LIN {X 0,Y 418.284,Z 298.384,A -85,B 0,C 180,E1 -10098.617,E2 -10098.617} C_VEL
LIN {X 0,Y 418.234,Z 298.38,A -85,B 0,C 180,E1 -10101.696,E2 -10101.696} C_VEL
LIN {X 0,Y 418.285,Z 298.377,A -85,B 0,C 180,E1 -10104.864,E2 -10104.864} C_VEL
LIN {X 0,Y 418.292,Z 298.377,A -85,B 0,C 180,E1 -10108.063,E2 -10108.063} C_VEL
LIN {X 0,Y 418.212,Z 298.39,A -85,B 0,C 180,E1 -10111.396,E2 -10111.396} C_VEL
LIN {X 0,Y 418.265,Z 298.378,A -85,B 0,C 180,E1 -10114.58,E2 -10114.58} C_VEL
LIN {X 0,Y 418.228,Z 298.385,A -85,B 0,C 180,E1 -10117.833,E2 -10117.833} C_VEL
LIN {X 0,Y 418.223,Z 298.387,A -85,B 0,C 180,E1 -10120.948,E2 -10120.948} C_VEL
LIN {X 0,Y 418.211,Z 298.392,A -85,B 0,C 180,E1 -10123.729,E2 -10123.729} C_VEL
LIN {X 0,Y 418.21,Z 298.388,A -85,B 0,C 180,E1 -10126.449,E2 -10126.449} C_VEL
LIN {X 0,Y 418.225,Z 298.389,A -85,B 0,C 180,E1 -10129.13,E2 -10129.13} C_VEL
LIN {X 0,Y 418.228,Z 298.39,A -85,B 0,C 180,E1 -10132.167,E2 -10132.167} C_VEL
LIN {X 0,Y 418.268,Z 298.385,A -85,B 0,C 180,E1 -10135.42,E2 -10135.42} C_VEL
LIN {X 0,Y 418.214,Z 298.387,A -85,B 0,C 180,E1 -10138.604,E2 -10138.604} C_VEL
LIN {X 0,Y 418.318,Z 298.464,A -85,B 0,C 180,E1 -10141.802,E2 -10141.802} C_VEL
LIN {X 0,Y 420.837,Z 310.121,A -85,B 0,C 180,E1 -10144.397,E2 -10144.397} C_VEL
LIN {X 0,Y 421.67,Z 315.968,A -85,B 0,C 180,E1 -10145.637,E2 -10145.637} C_VEL
LIN {X 0,Y 420.417,Z 334.149,A -85,B 0,C 180,E1 -10149.192,E2 -10149.192} C_VEL
LIN {X 0,Y 419.964,Z 341.407,A -85,B 0,C 180,E1 -10150.586,E2 -10150.586} C_VEL
LIN {X 0,Y 423.935,Z 364.685,A -85,B 0,C 180,E1 -10151.22,E2 -10151.22} C_VEL
LIN {X 0,Y 424.4,Z 369.391,A -85,B 0,C 180,E1 -10151.329,E2 -10151.329} C_VEL
LIN {X 0,Y 423.4,Z 449.942,A -85,B 0,C 180,E1 -10152.74,E2 -10152.74} C_VEL
LIN {X 0,Y 422.877,Z 463.116,A -85,B 0,C 180,E1 -10153.153,E2 -10153.153} C_VEL
LIN {X 0,Y 422.172,Z 475.789,A -85,B 0,C 180,E1 -10153.746,E2 -10153.746} C_VEL
LIN {X 0,Y 421.379,Z 487.877,A -85,B 0,C 180,E1 -10154.522,E2 -10154.522} C_VEL
LIN {X 0,Y 420.519,Z 499.381,A -85,B 0,C 180,E1 -10155.481,E2 -10155.481} C_VEL
LIN {X 0,Y 419.752,Z 509.766,A -85,B 0,C 180,E1 -10156.566,E2 -10156.566} C_VEL
LIN {X 0,Y 419.108,Z 518.281,A -85,B 0,C 180,E1 -10157.654,E2 -10157.654} C_VEL
LIN {X 0,Y 418.408,Z 526.153,A -85,B 0,C 180,E1 -10158.862,E2 -10158.862} C_VEL
LIN {X 0,Y 417.839,Z 533.861,A -85,B 0,C 180,E1 -10160.316,E2 -10160.316} C_VEL
LIN {X 0,Y 417.462,Z 540.067,A -85,B 0,C 180,E1 -10161.772,E2 -10161.772} C_VEL
LIN {X 0,Y 417.234,Z 545.013,A -85,B 0,C 180,E1 -10163.228,E2 -10163.228} C_VEL
LIN {X 0,Y 417.121,Z 548.84,A -85,B 0,C 180,E1 -10164.682,E2 -10164.682} C_VEL
LIN {X 0,Y 417.015,Z 551.649,A -85,B 0,C 180,E1 -10166.134,E2 -10166.134} C_VEL
LIN {X 0,Y 417.069,Z 553.924,A -85,B 0,C 180,E1 -10168.068,E2 -10168.068} C_VEL
LIN {X 0,Y 417.013,Z 554.464,A -85,B 0,C 180,E1 -10169.034,E2 -10169.034} C_VEL
LIN {X 0,Y 417.027,Z 554.573,A -85,B 0,C 180,E1 -10169.999,E2 -10169.999} C_VEL
LIN {X 0,Y 417.072,Z 553.622,A -85,B 0,C 180,E1 -10171.931,E2 -10171.931} C_VEL
LIN {X 0,Y 417.06,Z 552.553,A -85,B 0,C 180,E1 -10172.897,E2 -10172.897} C_VEL
LIN {X 0,Y 417.017,Z 551.024,A -85,B 0,C 180,E1 -10173.865,E2 -10173.865} C_VEL
LIN {X 0,Y 417.12,Z 547.943,A -85,B 0,C 180,E1 -10175.316,E2 -10175.316} C_VEL
LIN {X 0,Y 417.23,Z 543.788,A -85,B 0,C 180,E1 -10176.771,E2 -10176.771} C_VEL
LIN {X 0,Y 417.492,Z 537.427,A -85,B 0,C 180,E1 -10178.469,E2 -10178.469} C_VEL
LIN {X 0,Y 417.857,Z 530.492,A -85,B 0,C 180,E1 -10179.926,E2 -10179.926} C_VEL
LIN {X 0,Y 418.284,Z 523.404,A -85,B 0,C 180,E1 -10181.14,E2 -10181.14} C_VEL
LIN {X 0,Y 418.883,Z 514.854,A -85,B 0,C 180,E1 -10182.351,E2 -10182.351} C_VEL
LIN {X 0,Y 419.561,Z 504.271,A -85,B 0,C 180,E1 -10183.562,E2 -10183.562} C_VEL
LIN {X 0,Y 420.202,Z 493.786,A -85,B 0,C 180,E1 -10184.529,E2 -10184.529} C_VEL
LIN {X 0,Y 420.853,Z 482.263,A -85,B 0,C 180,E1 -10185.372,E2 -10185.372} C_VEL
LIN {X 0,Y 421.525,Z 470.346,A -85,B 0,C 180,E1 -10186.029,E2 -10186.029} C_VEL
LIN {X 0,Y 421.993,Z 458.396,A -85,B 0,C 180,E1 -10186.508,E2 -10186.508} C_VEL
LIN {X 0,Y 422.351,Z 445.617,A -85,B 0,C 180,E1 -10186.836,E2 -10186.836} C_VEL
LIN {X 0,Y 423.12,Z 367.397,A -85,B 0,C 180,E1 -10188.171,E2 -10188.171} C_VEL
LIN {X 0,Y 419.362,Z 341.793,A -85,B 0,C 180,E1 -10188.764,E2 -10188.764} C_VEL
LIN {X 0,Y 420.312,Z 325.648,A -85,B 0,C 180,E1 -10191.84,E2 -10191.84} C_VEL
LIN {X 0,Y 421.019,Z 313.701,A -85,B 0,C 180,E1 -10194.139,E2 -10194.139} C_VEL
LIN {X 0,Y 419.772,Z 305.575,A -85,B 0,C 180,E1 -10195.803,E2 -10195.803} C_VEL
LIN {X 0,Y 418.343,Z 298.377,A -85,B 0,C 180,E1 -10197.328,E2 -10197.328} C_VEL
LIN {X 0,Y 418.236,Z 298.384,A -85,B 0,C 180,E1 -10201.019,E2 -10201.019} C_VEL
LIN {X 0,Y 418.246,Z 298.384,A -85,B 0,C 180,E1 -10203.676,E2 -10203.676} C_VEL
LIN {X 0,Y 418.236,Z 298.383,A -85,B 0,C 180,E1 -10207.223,E2 -10207.223} C_VEL
LIN {X 0,Y 418.24,Z 298.383,A -85,B 0,C 180,E1 -10209.682,E2 -10209.682} C_VEL
LIN {X 0,Y 418.225,Z 298.391,A -85,B 0,C 180,E1 -10212.32,E2 -10212.32} C_VEL
LIN {X 0,Y 418.234,Z 298.384,A -85,B 0,C 180,E1 -10215.108,E2 -10215.108} C_VEL
LIN {X 0,Y 418.237,Z 298.383,A -85,B 0,C 180,E1 -10217.766,E2 -10217.766} C_VEL
LIN {X 0,Y 418.254,Z 298.389,A -85,B 0,C 180,E1 -10220.617,E2 -10220.617} C_VEL
LIN {X 0,Y 418.239,Z 298.383,A -85,B 0,C 180,E1 -10223.975,E2 -10223.975} C_VEL
LIN {X 0,Y 418.254,Z 298.384,A -85,B 0,C 180,E1 -10227.155,E2 -10227.155} C_VEL
LIN {X 0,Y 418.268,Z 298.386,A -85,B 0,C 180,E1 -10230.838,E2 -10230.838} C_VEL
LIN {X 0,Y 418.263,Z 298.38,A -85,B 0,C 180,E1 -10234.095,E2 -10234.095} C_VEL
LIN {X 0,Y 418.229,Z 298.389,A -85,B 0,C 180,E1 -10237.263,E2 -10237.263} C_VEL
LIN {X 0,Y 418.274,Z 298.378,A -85,B 0,C 180,E1 -10240.364,E2 -10240.364} C_VEL
LIN {X 0,Y 418.308,Z 298.38,A -85,B 0,C 180,E1 -10243.404,E2 -10243.404} C_VEL
LIN {X 0,Y 418.337,Z 298.374,A -85,B 0,C 180,E1 -10246.999,E2 -10246.999} C_VEL
LIN {X 0,Y 418.333,Z 298.371,A -85,B 0,C 180,E1 -10250.328,E2 -10250.328} C_VEL
LIN {X 0,Y 418.504,Z 298.35,A -85,B 0,C 180,E1 -10252.279,E2 -10252.279} C_VEL
LIN {X 0,Y 418.503,Z 298.35,A -85,B 0,C 180,E1 -10254.217,E2 -10254.217} C_VEL
LIN {X 0,Y 418.534,Z 298.348,A -85,B 0,C 180,E1 -10258.075,E2 -10258.075} C_VEL
LIN {X 0,Y 418.662,Z 298.334,A -85,B 0,C 180,E1 -10260,E2 -10260} C_VEL
LIN {X 0,Y 418.501,Z 298.35,A -85,B 0,C 180,E1 -10262.888,E2 -10262.888} C_VEL
LIN {X 0,Y 418.448,Z 298.357,A -85,B 0,C 180,E1 -10266.523,E2 -10266.523} C_VEL
LIN {X 0,Y 418.331,Z 298.376,A -85,B 0,C 180,E1 -10269.672,E2 -10269.672} C_VEL
LIN {X 0,Y 418.337,Z 298.37,A -85,B 0,C 180,E1 -10273.001,E2 -10273.001} C_VEL
LIN {X 0,Y 418.311,Z 298.375,A -85,B 0,C 180,E1 -10276.739,E2 -10276.739} C_VEL
LIN {X 0,Y 418.262,Z 298.383,A -85,B 0,C 180,E1 -10279.791,E2 -10279.791} C_VEL
LIN {X 0,Y 418.223,Z 298.387,A -85,B 0,C 180,E1 -10282.737,E2 -10282.737} C_VEL
LIN {X 0,Y 418.253,Z 298.383,A -85,B 0,C 180,E1 -10285.905,E2 -10285.905} C_VEL
LIN {X 0,Y 418.261,Z 298.381,A -85,B 0,C 180,E1 -10289.105,E2 -10289.105} C_VEL
LIN {X 0,Y 418.25,Z 298.385,A -85,B 0,C 180,E1 -10292.845,E2 -10292.845} C_VEL
LIN {X 0,Y 418.238,Z 298.386,A -85,B 0,C 180,E1 -10296.239,E2 -10296.239} C_VEL
LIN {X 0,Y 418.194,Z 298.388,A -85,B 0,C 180,E1 -10299.689,E2 -10299.689} C_VEL
LIN {X 0,Y 418.215,Z 298.388,A -85,B 0,C 180,E1 -10302.321,E2 -10302.321} C_VEL
LIN {X 0,Y 418.23,Z 298.388,A -85,B 0,C 180,E1 -10305.11,E2 -10305.11} C_VEL
LIN {X 0,Y 418.218,Z 298.385,A -85,B 0,C 180,E1 -10307.766,E2 -10307.766} C_VEL
LIN {X 0,Y 418.236,Z 298.385,A -85,B 0,C 180,E1 -10311.558,E2 -10311.558} C_VEL
LIN {X 0,Y 418.254,Z 298.389,A -85,B 0,C 180,E1 -10315.16,E2 -10315.16} C_VEL
LIN {X 0,Y 418.242,Z 298.387,A -85,B 0,C 180,E1 -10317.473,E2 -10317.473} C_VEL
LIN {X 0,Y 418.257,Z 298.383,A -85,B 0,C 180,E1 -10320.899,E2 -10320.899} C_VEL
LIN {X 0,Y 418.216,Z 298.386,A -85,B 0,C 180,E1 -10324.093,E2 -10324.093} C_VEL
LIN {X 0,Y 418.226,Z 298.389,A -85,B 0,C 180,E1 -10327.264,E2 -10327.264} C_VEL
LIN {X 0,Y 418.283,Z 298.377,A -85,B 0,C 180,E1 -10330.365,E2 -10330.365} C_VEL
LIN {X 0,Y 418.316,Z 298.378,A -85,B 0,C 180,E1 -10333.406,E2 -10333.406} C_VEL
LIN {X 0,Y 418.346,Z 298.37,A -85,B 0,C 180,E1 -10337.001,E2 -10337.001} C_VEL
LIN {X 0,Y 418.318,Z 298.378,A -85,B 0,C 180,E1 -10340.329,E2 -10340.329} C_VEL
LIN {X 0,Y 418.433,Z 298.431,A -85,B 0,C 180,E1 -10342.15,E2 -10342.15} C_VEL
LIN {X 0,Y 419.779,Z 306.465,A -85,B 0,C 180,E1 -10343.994,E2 -10343.994} C_VEL
LIN {X 0,Y 419.625,Z 312.565,A -85,B 0,C 180,E1 -10345.319,E2 -10345.319} C_VEL
LIN {X 0,Y 423.458,Z 333.219,A -85,B 0,C 180,E1 -10345.834,E2 -10345.834} C_VEL
LIN {X 0,Y 422.406,Z 420.671,A -85,B 0,C 180,E1 -10347.346,E2 -10347.346} C_VEL
LIN {X 0,Y 422.186,Z 427.807,A -85,B 0,C 180,E1 -10347.552,E2 -10347.552} C_VEL
LIN {X 0,Y 421.371,Z 433.517,A -85,B 0,C 180,E1 -10347.735,E2 -10347.735} C_VEL
LIN {X 0,Y 418.244,Z 442.663,A -85,B 0,C 180,E1 -10348.05,E2 -10348.05} C_VEL
LIN {X 0,Y 415.058,Z 451.531,A -85,B 0,C 180,E1 -10348.471,E2 -10348.471} C_VEL
LIN {X 0,Y 414.153,Z 456.798,A -85,B 0,C 180,E1 -10348.816,E2 -10348.816} C_VEL
LIN {X 0,Y 413.498,Z 468.178,A -85,B 0,C 180,E1 -10349.757,E2 -10349.757} C_VEL
LIN {X 0,Y 412.779,Z 478.733,A -85,B 0,C 180,E1 -10350.854,E2 -10350.854} C_VEL
LIN {X 0,Y 412.151,Z 487.368,A -85,B 0,C 180,E1 -10351.955,E2 -10351.955} C_VEL
LIN {X 0,Y 411.564,Z 495.326,A -85,B 0,C 180,E1 -10353.182,E2 -10353.182} C_VEL
LIN {X 0,Y 411.026,Z 503.123,A -85,B 0,C 180,E1 -10354.659,E2 -10354.659} C_VEL
LIN {X 0,Y 410.673,Z 509.679,A -85,B 0,C 180,E1 -10356.23,E2 -10356.23} C_VEL
LIN {X 0,Y 410.333,Z 515.036,A -85,B 0,C 180,E1 -10357.876,E2 -10357.876} C_VEL
LIN {X 0,Y 410.103,Z 518.7,A -85,B 0,C 180,E1 -10359.37,E2 -10359.37} C_VEL
LIN {X 0,Y 409.992,Z 521.335,A -85,B 0,C 180,E1 -10360.869,E2 -10360.869} C_VEL
LIN {X 0,Y 409.922,Z 522.9,A -85,B 0,C 180,E1 -10362.244,E2 -10362.244} C_VEL
LIN {X 0,Y 409.815,Z 523.749,A -85,B 0,C 180,E1 -10363.892,E2 -10363.892} C_VEL
LIN {X 0,Y 409.852,Z 523.728,A -85,B 0,C 180,E1 -10364.905,E2 -10364.905} C_VEL
LIN {X 0,Y 409.924,Z 523.045,A -85,B 0,C 180,E1 -10366.239,E2 -10366.239} C_VEL
LIN {X 0,Y 410.002,Z 521.082,A -85,B 0,C 180,E1 -10367.972,E2 -10367.972} C_VEL
LIN {X 0,Y 410.314,Z 518.063,A -85,B 0,C 180,E1 -10369.599,E2 -10369.599} C_VEL
LIN {X 0,Y 410.584,Z 514.287,A -85,B 0,C 180,E1 -10371.067,E2 -10371.067} C_VEL
LIN {X 0,Y 411.065,Z 508.427,A -85,B 0,C 180,E1 -10372.798,E2 -10372.798} C_VEL
LIN {X 0,Y 411.725,Z 501.106,A -85,B 0,C 180,E1 -10374.453,E2 -10374.453} C_VEL
LIN {X 0,Y 412.316,Z 494.236,A -85,B 0,C 180,E1 -10375.709,E2 -10375.709} C_VEL
LIN {X 0,Y 413.089,Z 485.156,A -85,B 0,C 180,E1 -10377.072,E2 -10377.072} C_VEL
LIN {X 0,Y 413.946,Z 475.508,A -85,B 0,C 180,E1 -10378.236,E2 -10378.236} C_VEL
LIN {X 0,Y 414.832,Z 464.643,A -85,B 0,C 180,E1 -10379.288,E2 -10379.288} C_VEL
LIN {X 0,Y 415.607,Z 452.692,A -85,B 0,C 180,E1 -10380.204,E2 -10380.204} C_VEL
LIN {X 0,Y 416.266,Z 440.132,A -85,B 0,C 180,E1 -10380.924,E2 -10380.924} C_VEL
LIN {X 0,Y 416.758,Z 427.18,A -85,B 0,C 180,E1 -10381.448,E2 -10381.448} C_VEL
LIN {X 0,Y 417.031,Z 413.94,A -85,B 0,C 180,E1 -10381.779,E2 -10381.779} C_VEL
LIN {X 0,Y 418.276,Z 334.084,A -85,B 0,C 180,E1 -10383.17,E2 -10383.17} C_VEL
LIN {X 0,Y 414.67,Z 317.421,A -85,B 0,C 180,E1 -10383.684,E2 -10383.684} C_VEL
LIN {X 0,Y 413.565,Z 312.818,A -85,B 0,C 180,E1 -10383.857,E2 -10383.857} C_VEL
LIN {X 0,Y 413.337,Z 308.963,A -85,B 0,C 180,E1 -10384.723,E2 -10384.723} C_VEL
LIN {X 0,Y 411.204,Z 299.261,A -85,B 0,C 180,E1 -10387.085,E2 -10387.085} C_VEL
LIN {X 0,Y 411.182,Z 299.268,A -85,B 0,C 180,E1 -10390.504,E2 -10390.504} C_VEL
LIN {X 0,Y 411.175,Z 299.269,A -85,B 0,C 180,E1 -10393.134,E2 -10393.134} C_VEL
LIN {X 0,Y 411.17,Z 299.269,A -85,B 0,C 180,E1 -10395.881,E2 -10395.881} C_VEL
LIN {X 0,Y 411.167,Z 299.273,A -85,B 0,C 180,E1 -10398.771,E2 -10398.771} C_VEL
LIN {X 0,Y 411.208,Z 299.259,A -85,B 0,C 180,E1 -10401.831,E2 -10401.831} C_VEL
LIN {X 0,Y 411.212,Z 299.265,A -85,B 0,C 180,E1 -10405.121,E2 -10405.121} C_VEL
LIN {X 0,Y 411.167,Z 299.265,A -85,B 0,C 180,E1 -10408.003,E2 -10408.003} C_VEL
LIN {X 0,Y 411.219,Z 299.262,A -85,B 0,C 180,E1 -10411.41,E2 -10411.41} C_VEL
LIN {X 0,Y 411.239,Z 299.257,A -85,B 0,C 180,E1 -10413.619,E2 -10413.619} C_VEL
LIN {X 0,Y 411.204,Z 299.26,A -85,B 0,C 180,E1 -10416.852,E2 -10416.852} C_VEL
LIN {X 0,Y 411.215,Z 299.256,A -85,B 0,C 180,E1 -10420.05,E2 -10420.05} C_VEL
LIN {X 0,Y 411.264,Z 299.255,A -85,B 0,C 180,E1 -10423.131,E2 -10423.131} C_VEL
LIN {X 0,Y 411.306,Z 299.245,A -85,B 0,C 180,E1 -10426.896,E2 -10426.896} C_VEL
LIN {X 0,Y 411.293,Z 299.242,A -85,B 0,C 180,E1 -10430.161,E2 -10430.161} C_VEL
LIN {X 0,Y 411.483,Z 299.228,A -85,B 0,C 180,E1 -10432.147,E2 -10432.147} C_VEL
LIN {X 0,Y 411.472,Z 299.226,A -85,B 0,C 180,E1 -10434.118,E2 -10434.118} C_VEL
LIN {X 0,Y 411.511,Z 299.227,A -85,B 0,C 180,E1 -10438.043,E2 -10438.043} C_VEL
LIN {X 0,Y 411.64,Z 299.203,A -85,B 0,C 180,E1 -10440,E2 -10440} C_VEL
LIN {X 0,Y 411.458,Z 299.227,A -85,B 0,C 180,E1 -10442.937,E2 -10442.937} C_VEL
LIN {X 0,Y 411.458,Z 299.224,A -85,B 0,C 180,E1 -10446.867,E2 -10446.867} C_VEL
LIN {X 0,Y 411.354,Z 299.241,A -85,B 0,C 180,E1 -10448.845,E2 -10448.845} C_VEL
LIN {X 0,Y 411.283,Z 299.242,A -85,B 0,C 180,E1 -10451.833,E2 -10451.833} C_VEL
LIN {X 0,Y 411.26,Z 299.251,A -85,B 0,C 180,E1 -10454.853,E2 -10454.853} C_VEL
LIN {X 0,Y 411.253,Z 299.253,A -85,B 0,C 180,E1 -10457.915,E2 -10457.915} C_VEL
LIN {X 0,Y 411.197,Z 299.258,A -85,B 0,C 180,E1 -10461.034,E2 -10461.034} C_VEL
LIN {X 0,Y 411.221,Z 299.26,A -85,B 0,C 180,E1 -10464.216,E2 -10464.216} C_VEL
LIN {X 0,Y 411.26,Z 299.254,A -85,B 0,C 180,E1 -10467.478,E2 -10467.478} C_VEL
LIN {X 0,Y 411.19,Z 299.261,A -85,B 0,C 180,E1 -10470.848,E2 -10470.848} C_VEL
LIN {X 0,Y 411.205,Z 299.255,A -85,B 0,C 180,E1 -10474.334,E2 -10474.334} C_VEL
LIN {X 0,Y 411.194,Z 299.261,A -85,B 0,C 180,E1 -10477.974,E2 -10477.974} C_VEL
LIN {X 0,Y 411.165,Z 299.268,A -85,B 0,C 180,E1 -10481.228,E2 -10481.228} C_VEL
LIN {X 0,Y 411.177,Z 299.265,A -85,B 0,C 180,E1 -10484.49,E2 -10484.49} C_VEL
LIN {X 0,Y 411.179,Z 299.265,A -85,B 0,C 180,E1 -10488.195,E2 -10488.195} C_VEL
LIN {X 0,Y 411.213,Z 299.255,A -85,B 0,C 180,E1 -10490.775,E2 -10490.775} C_VEL
LIN {X 0,Y 411.2,Z 299.261,A -85,B 0,C 180,E1 -10494.471,E2 -10494.471} C_VEL
LIN {X 0,Y 411.21,Z 299.258,A -85,B 0,C 180,E1 -10496.873,E2 -10496.873} C_VEL
LIN {X 0,Y 411.236,Z 299.258,A -85,B 0,C 180,E1 -10500.644,E2 -10500.644} C_VEL
LIN {X 0,Y 411.283,Z 299.335,A -85,B 0,C 180,E1 -10501.453,E2 -10501.453} C_VEL
LIN {X 0,Y 413.867,Z 311.218,A -85,B 0,C 180,E1 -10504.16,E2 -10504.16} C_VEL
LIN {X 0,Y 414.798,Z 317.271,A -85,B 0,C 180,E1 -10505.473,E2 -10505.473} C_VEL
LIN {X 0,Y 413.555,Z 334.145,A -85,B 0,C 180,E1 -10508.83,E2 -10508.83} C_VEL
LIN {X 0,Y 413.096,Z 341.021,A -85,B 0,C 180,E1 -10510.184,E2 -10510.184} C_VEL
LIN {X 0,Y 417.111,Z 363.869,A -85,B 0,C 180,E1 -10510.841,E2 -10510.841} C_VEL
LIN {X 0,Y 417.802,Z 369.66,A -85,B 0,C 180,E1 -10510.984,E2 -10510.984} C_VEL
LIN {X 0,Y 416.721,Z 450.224,A -85,B 0,C 180,E1 -10512.422,E2 -10512.422} C_VEL
LIN {X 0,Y 416.167,Z 463.217,A -85,B 0,C 180,E1 -10512.842,E2 -10512.842} C_VEL
LIN {X 0,Y 415.405,Z 476.34,A -85,B 0,C 180,E1 -10513.474,E2 -10513.474} C_VEL
LIN {X 0,Y 414.562,Z 488.193,A -85,B 0,C 180,E1 -10514.261,E2 -10514.261} C_VEL
LIN {X 0,Y 413.652,Z 499.591,A -85,B 0,C 180,E1 -10515.235,E2 -10515.235} C_VEL
LIN {X 0,Y 412.832,Z 509.89,A -85,B 0,C 180,E1 -10516.337,E2 -10516.337} C_VEL
LIN {X 0,Y 412.152,Z 518.328,A -85,B 0,C 180,E1 -10517.442,E2 -10517.442} C_VEL
LIN {X 0,Y 411.301,Z 527.498,A -85,B 0,C 180,E1 -10518.916,E2 -10518.916} C_VEL
LIN {X 0,Y 410.744,Z 534.898,A -85,B 0,C 180,E1 -10520.396,E2 -10520.396} C_VEL
LIN {X 0,Y 410.322,Z 541.736,A -85,B 0,C 180,E1 -10522.124,E2 -10522.124} C_VEL
LIN {X 0,Y 410.043,Z 546.698,A -85,B 0,C 180,E1 -10523.774,E2 -10523.774} C_VEL
LIN {X 0,Y 410.018,Z 549.718,A -85,B 0,C 180,E1 -10525.083,E2 -10525.083} C_VEL
LIN {X 0,Y 409.928,Z 552.761,A -85,B 0,C 180,E1 -10527.051,E2 -10527.051} C_VEL
LIN {X 0,Y 409.996,Z 553.691,A -85,B 0,C 180,E1 -10528.035,E2 -10528.035} C_VEL
LIN {X 0,Y 409.938,Z 554.209,A -85,B 0,C 180,E1 -10529.017,E2 -10529.017} C_VEL
LIN {X 0,Y 409.948,Z 554.302,A -85,B 0,C 180,E1 -10529.999,E2 -10529.999} C_VEL
LIN {X 0,Y 410,Z 553.326,A -85,B 0,C 180,E1 -10531.964,E2 -10531.964} C_VEL
LIN {X 0,Y 409.959,Z 552.234,A -85,B 0,C 180,E1 -10532.947,E2 -10532.947} C_VEL
LIN {X 0,Y 409.936,Z 550.687,A -85,B 0,C 180,E1 -10533.931,E2 -10533.931} C_VEL
LIN {X 0,Y 410.017,Z 547.576,A -85,B 0,C 180,E1 -10535.409,E2 -10535.409} C_VEL
LIN {X 0,Y 410.162,Z 543.392,A -85,B 0,C 180,E1 -10536.888,E2 -10536.888} C_VEL
LIN {X 0,Y 410.423,Z 536.996,A -85,B 0,C 180,E1 -10538.616,E2 -10538.616} C_VEL
LIN {X 0,Y 410.799,Z 530.022,A -85,B 0,C 180,E1 -10540.099,E2 -10540.099} C_VEL
LIN {X 0,Y 411.414,Z 521.274,A -85,B 0,C 180,E1 -10541.578,E2 -10541.578} C_VEL
LIN {X 0,Y 412.001,Z 512.298,A -85,B 0,C 180,E1 -10542.811,E2 -10542.811} C_VEL
LIN {X 0,Y 412.648,Z 502.786,A -85,B 0,C 180,E1 -10543.881,E2 -10543.881} C_VEL
LIN {X 0,Y 413.361,Z 491.551,A -85,B 0,C 180,E1 -10544.9,E2 -10544.9} C_VEL
LIN {X 0,Y 414.111,Z 479.331,A -85,B 0,C 180,E1 -10545.755,E2 -10545.755} C_VEL
LIN {X 0,Y 414.783,Z 466.548,A -85,B 0,C 180,E1 -10546.423,E2 -10546.423} C_VEL
LIN {X 0,Y 415.318,Z 453.863,A -85,B 0,C 180,E1 -10546.876,E2 -10546.876} C_VEL
LIN {X 0,Y 415.597,Z 435.872,A -85,B 0,C 180,E1 -10547.244,E2 -10547.244} C_VEL
LIN {X 0,Y 416.181,Z 367.386,A -85,B 0,C 180,E1 -10548.432,E2 -10548.432} C_VEL
LIN {X 0,Y 412.412,Z 341.451,A -85,B 0,C 180,E1 -10549.06,E2 -10549.06} C_VEL
LIN {X 0,Y 413.329,Z 326.457,A -85,B 0,C 180,E1 -10551.966,E2 -10551.966} C_VEL
LIN {X 0,Y 414.035,Z 314.493,A -85,B 0,C 180,E1 -10554.306,E2 -10554.306} C_VEL
LIN {X 0,Y 412.412,Z 304.976,A -85,B 0,C 180,E1 -10556.299,E2 -10556.299} C_VEL
LIN {X 0,Y 411.319,Z 299.251,A -85,B 0,C 180,E1 -10557.541,E2 -10557.541} C_VEL
LIN {X 0,Y 411.18,Z 299.263,A -85,B 0,C 180,E1 -10561.283,E2 -10561.283} C_VEL
LIN {X 0,Y 411.203,Z 299.265,A -85,B 0,C 180,E1 -10564.332,E2 -10564.332} C_VEL
LIN {X 0,Y 411.188,Z 299.265,A -85,B 0,C 180,E1 -10567.973,E2 -10567.973} C_VEL
LIN {X 0,Y 411.158,Z 299.265,A -85,B 0,C 180,E1 -10571.227,E2 -10571.227} C_VEL
LIN {X 0,Y 411.172,Z 299.271,A -85,B 0,C 180,E1 -10574.489,E2 -10574.489} C_VEL
LIN {X 0,Y 411.173,Z 299.266,A -85,B 0,C 180,E1 -10578.194,E2 -10578.194} C_VEL
LIN {X 0,Y 411.218,Z 299.263,A -85,B 0,C 180,E1 -10580.776,E2 -10580.776} C_VEL
LIN {X 0,Y 411.193,Z 299.265,A -85,B 0,C 180,E1 -10584.471,E2 -10584.471} C_VEL
LIN {X 0,Y 411.165,Z 299.264,A -85,B 0,C 180,E1 -10588.003,E2 -10588.003} C_VEL
LIN {X 0,Y 411.216,Z 299.259,A -85,B 0,C 180,E1 -10591.41,E2 -10591.41} C_VEL
LIN {X 0,Y 411.228,Z 299.26,A -85,B 0,C 180,E1 -10594.706,E2 -10594.706} C_VEL
LIN {X 0,Y 411.197,Z 299.26,A -85,B 0,C 180,E1 -10597.913,E2 -10597.913} C_VEL
LIN {X 0,Y 411.216,Z 299.264,A -85,B 0,C 180,E1 -10601.051,E2 -10601.051} C_VEL
LIN {X 0,Y 411.246,Z 299.254,A -85,B 0,C 180,E1 -10604.131,E2 -10604.131} C_VEL
LIN {X 0,Y 411.294,Z 299.253,A -85,B 0,C 180,E1 -10607.165,E2 -10607.165} C_VEL
LIN {X 0,Y 411.285,Z 299.249,A -85,B 0,C 180,E1 -10610.161,E2 -10610.161} C_VEL
LIN {X 0,Y 411.451,Z 299.231,A -85,B 0,C 180,E1 -10613.133,E2 -10613.133} C_VEL
LIN {X 0,Y 411.301,Z 299.249,A -85,B 0,C 180,E1 -10615.099,E2 -10615.099} C_VEL
LIN {X 0,Y 411.503,Z 299.224,A -85,B 0,C 180,E1 -10618.043,E2 -10618.043} C_VEL
LIN {X 0,Y 411.632,Z 299.209,A -85,B 0,C 180,E1 -10620,E2 -10620} C_VEL
LIN {X 0,Y 411.457,Z 299.228,A -85,B 0,C 180,E1 -10622.937,E2 -10622.937} C_VEL
LIN {X 0,Y 411.414,Z 299.233,A -85,B 0,C 180,E1 -10626.868,E2 -10626.868} C_VEL
LIN {X 0,Y 411.283,Z 299.256,A -85,B 0,C 180,E1 -10629.839,E2 -10629.839} C_VEL
LIN {X 0,Y 411.296,Z 299.247,A -85,B 0,C 180,E1 -10633.104,E2 -10633.104} C_VEL
LIN {X 0,Y 411.255,Z 299.253,A -85,B 0,C 180,E1 -10636.87,E2 -10636.87} C_VEL
LIN {X 0,Y 411.222,Z 299.262,A -85,B 0,C 180,E1 -10639.987,E2 -10639.987} C_VEL
LIN {X 0,Y 411.187,Z 299.261,A -85,B 0,C 180,E1 -10643.149,E2 -10643.149} C_VEL
LIN {X 0,Y 411.225,Z 299.264,A -85,B 0,C 180,E1 -10646.382,E2 -10646.382} C_VEL
LIN {X 0,Y 411.193,Z 299.261,A -85,B 0,C 180,E1 -10649.714,E2 -10649.714} C_VEL
LIN {X 0,Y 411.199,Z 299.261,A -85,B 0,C 180,E1 -10653.157,E2 -10653.157} C_VEL
LIN {X 0,Y 411.185,Z 299.268,A -85,B 0,C 180,E1 -10656.553,E2 -10656.553} C_VEL
LIN {X 0,Y 411.163,Z 299.264,A -85,B 0,C 180,E1 -10659.721,E2 -10659.721} C_VEL
LIN {X 0,Y 411.164,Z 299.268,A -85,B 0,C 180,E1 -10663.135,E2 -10663.135} C_VEL
LIN {X 0,Y 411.159,Z 299.264,A -85,B 0,C 180,E1 -10665.883,E2 -10665.883} C_VEL
LIN {X 0,Y 411.146,Z 299.271,A -85,B 0,C 180,E1 -10668.775,E2 -10668.775} C_VEL
LIN {X 0,Y 411.183,Z 299.262,A -85,B 0,C 180,E1 -10672.027,E2 -10672.027} C_VEL
LIN {X 0,Y 411.201,Z 299.261,A -85,B 0,C 180,E1 -10675.667,E2 -10675.667} C_VEL
LIN {X 0,Y 411.186,Z 299.268,A -85,B 0,C 180,E1 -10679.153,E2 -10679.153} C_VEL
LIN {X 0,Y 411.17,Z 299.27,A -85,B 0,C 180,E1 -10681.408,E2 -10681.408} C_VEL
LIN {X 0,Y 411.186,Z 299.263,A -85,B 0,C 180,E1 -10684.942,E2 -10684.942} C_VEL
LIN {X 0,Y 411.202,Z 299.262,A -85,B 0,C 180,E1 -10687.914,E2 -10687.914} C_VEL
LIN {X 0,Y 411.218,Z 299.259,A -85,B 0,C 180,E1 -10691.052,E2 -10691.052} C_VEL
LIN {X 0,Y 411.252,Z 299.255,A -85,B 0,C 180,E1 -10694.133,E2 -10694.133} C_VEL
LIN {X 0,Y 411.302,Z 299.248,A -85,B 0,C 180,E1 -10697.167,E2 -10697.167} C_VEL
LIN {X 0,Y 411.272,Z 299.256,A -85,B 0,C 180,E1 -10700.162,E2 -10700.162} C_VEL
LIN {X 0,Y 411.4,Z 299.41,A -85,B 0,C 180,E1 -10701.985,E2 -10701.985} C_VEL
LIN {X 0,Y 412.787,Z 307.592,A -85,B 0,C 180,E1 -10703.892,E2 -10703.892} C_VEL
LIN {X 0,Y 412.664,Z 312.726,A -85,B 0,C 180,E1 -10705.024,E2 -10705.024} C_VEL
LIN {X 0,Y 416.636,Z 333.923,A -85,B 0,C 180,E1 -10705.58,E2 -10705.58} C_VEL
LIN {X 0,Y 415.565,Z 420.284,A -85,B 0,C 180,E1 -10707.093,E2 -10707.093} C_VEL
LIN {X 0,Y 415.154,Z 433.403,A -85,B 0,C 180,E1 -10707.515,E2 -10707.515} C_VEL
LIN {X 0,Y 414.727,Z 445.968,A -85,B 0,C 180,E1 -10708.119,E2 -10708.119} C_VEL
LIN {X 0,Y 414.153,Z 456.798,A -85,B 0,C 180,E1 -10708.816,E2 -10708.816} C_VEL
LIN {X 0,Y 413.225,Z 461.979,A -85,B 0,C 180,E1 -10709.193,E2 -10709.193} C_VEL
LIN {X 0,Y 409.865,Z 470.129,A -85,B 0,C 180,E1 -10709.83,E2 -10709.83} C_VEL
LIN {X 0,Y 406.486,Z 477.887,A -85,B 0,C 180,E1 -10710.558,E2 -10710.558} C_VEL
LIN {X 0,Y 405.52,Z 482.359,A -85,B 0,C 180,E1 -10711.083,E2 -10711.083} C_VEL
LIN {X 0,Y 404.788,Z 492.28,A -85,B 0,C 180,E1 -10712.488,E2 -10712.488} C_VEL
LIN {X 0,Y 404.165,Z 500.703,A -85,B 0,C 180,E1 -10713.989,E2 -10713.989} C_VEL
LIN {X 0,Y 403.657,Z 507.484,A -85,B 0,C 180,E1 -10715.496,E2 -10715.496} C_VEL
LIN {X 0,Y 403.403,Z 512.893,A -85,B 0,C 180,E1 -10717.005,E2 -10717.005} C_VEL
LIN {X 0,Y 403.138,Z 517.138,A -85,B 0,C 180,E1 -10718.522,E2 -10718.522} C_VEL
LIN {X 0,Y 402.915,Z 520.318,A -85,B 0,C 180,E1 -10720.046,E2 -10720.046} C_VEL
LIN {X 0,Y 402.88,Z 521.896,A -85,B 0,C 180,E1 -10721.064,E2 -10721.064} C_VEL
LIN {X 0,Y 402.828,Z 523.204,A -85,B 0,C 180,E1 -10722.308,E2 -10722.308} C_VEL
LIN {X 0,Y 402.747,Z 524.048,A -85,B 0,C 180,E1 -10724.141,E2 -10724.141} C_VEL
LIN {X 0,Y 402.78,Z 523.955,A -85,B 0,C 180,E1 -10725.173,E2 -10725.173} C_VEL
LIN {X 0,Y 402.839,Z 523.289,A -85,B 0,C 180,E1 -10726.353,E2 -10726.353} C_VEL
LIN {X 0,Y 402.96,Z 521.051,A -85,B 0,C 180,E1 -10728.297,E2 -10728.297} C_VEL
LIN {X 0,Y 403.272,Z 518.285,A -85,B 0,C 180,E1 -10729.765,E2 -10729.765} C_VEL
LIN {X 0,Y 403.601,Z 513.955,A -85,B 0,C 180,E1 -10731.45,E2 -10731.45} C_VEL
LIN {X 0,Y 404.095,Z 508.426,A -85,B 0,C 180,E1 -10733.066,E2 -10733.066} C_VEL
LIN {X 0,Y 404.742,Z 501.628,A -85,B 0,C 180,E1 -10734.629,E2 -10734.629} C_VEL
LIN {X 0,Y 405.419,Z 494.502,A -85,B 0,C 180,E1 -10735.958,E2 -10735.958} C_VEL
LIN {X 0,Y 406.196,Z 485.796,A -85,B 0,C 180,E1 -10737.291,E2 -10737.291} C_VEL
LIN {X 0,Y 407.113,Z 476.03,A -85,B 0,C 180,E1 -10738.499,E2 -10738.499} C_VEL
LIN {X 0,Y 408.018,Z 465.524,A -85,B 0,C 180,E1 -10739.542,E2 -10739.542} C_VEL
LIN {X 0,Y 408.894,Z 453.245,A -85,B 0,C 180,E1 -10740.506,E2 -10740.506} C_VEL
LIN {X 0,Y 409.541,Z 441.576,A -85,B 0,C 180,E1 -10741.201,E2 -10741.201} C_VEL
LIN {X 0,Y 410.062,Z 429.131,A -85,B 0,C 180,E1 -10741.732,E2 -10741.732} C_VEL
LIN {X 0,Y 410.397,Z 415.694,A -85,B 0,C 180,E1 -10742.097,E2 -10742.097} C_VEL
LIN {X 0,Y 411.687,Z 334.543,A -85,B 0,C 180,E1 -10743.539,E2 -10743.539} C_VEL
LIN {X 0,Y 407.641,Z 316.789,A -85,B 0,C 180,E1 -10744.114,E2 -10744.114} C_VEL
LIN {X 0,Y 406.745,Z 313.099,A -85,B 0,C 180,E1 -10744.258,E2 -10744.258} C_VEL
LIN {X 0,Y 405.676,Z 306.899,A -85,B 0,C 180,E1 -10745.734,E2 -10745.734} C_VEL
LIN {X 0,Y 404.167,Z 300.138,A -85,B 0,C 180,E1 -10747.444,E2 -10747.444} C_VEL
LIN {X 0,Y 404.15,Z 300.145,A -85,B 0,C 180,E1 -10750.08,E2 -10750.08} C_VEL
LIN {X 0,Y 404.155,Z 300.144,A -85,B 0,C 180,E1 -10753.084,E2 -10753.084} C_VEL
LIN {X 0,Y 404.15,Z 300.143,A -85,B 0,C 180,E1 -10755.926,E2 -10755.926} C_VEL
LIN {X 0,Y 404.122,Z 300.153,A -85,B 0,C 180,E1 -10758.635,E2 -10758.635} C_VEL
LIN {X 0,Y 404.157,Z 300.138,A -85,B 0,C 180,E1 -10761.492,E2 -10761.492} C_VEL
LIN {X 0,Y 404.186,Z 300.14,A -85,B 0,C 180,E1 -10764.984,E2 -10764.984} C_VEL
LIN {X 0,Y 404.143,Z 300.143,A -85,B 0,C 180,E1 -10768.554,E2 -10768.554} C_VEL
LIN {X 0,Y 404.197,Z 300.133,A -85,B 0,C 180,E1 -10772,E2 -10772} C_VEL
LIN {X 0,Y 404.179,Z 300.139,A -85,B 0,C 180,E1 -10775.334,E2 -10775.334} C_VEL
LIN {X 0,Y 404.139,Z 300.14,A -85,B 0,C 180,E1 -10778.581,E2 -10778.581} C_VEL
LIN {X 0,Y 404.211,Z 300.132,A -85,B 0,C 180,E1 -10781.762,E2 -10781.762} C_VEL
LIN {X 0,Y 404.206,Z 300.131,A -85,B 0,C 180,E1 -10784.882,E2 -10784.882} C_VEL
LIN {X 0,Y 404.256,Z 300.128,A -85,B 0,C 180,E1 -10787.958,E2 -10787.958} C_VEL
LIN {X 0,Y 404.434,Z 300.107,A -85,B 0,C 180,E1 -10792.1,E2 -10792.1} C_VEL
LIN {X 0,Y 404.421,Z 300.106,A -85,B 0,C 180,E1 -10794.015,E2 -10794.015} C_VEL
LIN {X 0,Y 404.48,Z 300.103,A -85,B 0,C 180,E1 -10798.008,E2 -10798.008} C_VEL
LIN {X 0,Y 404.609,Z 300.078,A -85,B 0,C 180,E1 -10800,E2 -10800} C_VEL
LIN {X 0,Y 404.416,Z 300.104,A -85,B 0,C 180,E1 -10802.988,E2 -10802.988} C_VEL
LIN {X 0,Y 404.41,Z 300.102,A -85,B 0,C 180,E1 -10806.987,E2 -10806.987} C_VEL
LIN {X 0,Y 404.257,Z 300.127,A -85,B 0,C 180,E1 -10810.012,E2 -10810.012} C_VEL
LIN {X 0,Y 404.267,Z 300.123,A -85,B 0,C 180,E1 -10813.211,E2 -10813.211} C_VEL
LIN {X 0,Y 404.216,Z 300.13,A -85,B 0,C 180,E1 -10817.007,E2 -10817.007} C_VEL
LIN {X 0,Y 404.164,Z 300.138,A -85,B 0,C 180,E1 -10820.352,E2 -10820.352} C_VEL
LIN {X 0,Y 404.164,Z 300.138,A -85,B 0,C 180,E1 -10823.575,E2 -10823.575} C_VEL
LIN {X 0,Y 404.184,Z 300.127,A -85,B 0,C 180,E1 -10825.766,E2 -10825.766} C_VEL
LIN {X 0,Y 404.196,Z 300.133,A -85,B 0,C 180,E1 -10828,E2 -10828} C_VEL
LIN {X 0,Y 404.14,Z 300.141,A -85,B 0,C 180,E1 -10831.558,E2 -10831.558} C_VEL
LIN {X 0,Y 404.184,Z 300.136,A -85,B 0,C 180,E1 -10835.016,E2 -10835.016} C_VEL
LIN {X 0,Y 404.153,Z 300.14,A -85,B 0,C 180,E1 -10838.757,E2 -10838.757} C_VEL
LIN {X 0,Y 404.124,Z 300.147,A -85,B 0,C 180,E1 -10841.6,E2 -10841.6} C_VEL
LIN {X 0,Y 404.147,Z 300.141,A -85,B 0,C 180,E1 -10844.522,E2 -10844.522} C_VEL
LIN {X 0,Y 404.138,Z 300.147,A -85,B 0,C 180,E1 -10847.296,E2 -10847.296} C_VEL
LIN {X 0,Y 404.171,Z 300.135,A -85,B 0,C 180,E1 -10849.955,E2 -10849.955} C_VEL
LIN {X 0,Y 404.138,Z 300.146,A -85,B 0,C 180,E1 -10853.125,E2 -10853.125} C_VEL
LIN {X 0,Y 404.148,Z 300.14,A -85,B 0,C 180,E1 -10856.188,E2 -10856.188} C_VEL
LIN {X 0,Y 404.148,Z 300.144,A -85,B 0,C 180,E1 -10859.715,E2 -10859.715} C_VEL
LIN {X 0,Y 404.216,Z 300.179,A -85,B 0,C 180,E1 -10861.081,E2 -10861.081} C_VEL
LIN {X 0,Y 406.916,Z 312.319,A -85,B 0,C 180,E1 -10863.911,E2 -10863.911} C_VEL
LIN {X 0,Y 407.923,Z 318.587,A -85,B 0,C 180,E1 -10865.304,E2 -10865.304} C_VEL
LIN {X 0,Y 406.635,Z 335.447,A -85,B 0,C 180,E1 -10868.718,E2 -10868.718} C_VEL
LIN {X 0,Y 406.293,Z 340.897,A -85,B 0,C 180,E1 -10869.793,E2 -10869.793} C_VEL
LIN {X 0,Y 410.702,Z 366.016,A -85,B 0,C 180,E1 -10870.523,E2 -10870.523} C_VEL
LIN {X 0,Y 411.207,Z 370.647,A -85,B 0,C 180,E1 -10870.638,E2 -10870.638} C_VEL
LIN {X 0,Y 410.06,Z 449.437,A -85,B 0,C 180,E1 -10872.063,E2 -10872.063} C_VEL
LIN {X 0,Y 409.514,Z 462.581,A -85,B 0,C 180,E1 -10872.49,E2 -10872.49} C_VEL
LIN {X 0,Y 408.72,Z 475.796,A -85,B 0,C 180,E1 -10873.131,E2 -10873.131} C_VEL
LIN {X 0,Y 407.882,Z 486.935,A -85,B 0,C 180,E1 -10873.868,E2 -10873.868} C_VEL
LIN {X 0,Y 406.873,Z 498.514,A -85,B 0,C 180,E1 -10874.855,E2 -10874.855} C_VEL
LIN {X 0,Y 405.979,Z 508.952,A -85,B 0,C 180,E1 -10875.974,E2 -10875.974} C_VEL
LIN {X 0,Y 405.218,Z 518.379,A -85,B 0,C 180,E1 -10877.224,E2 -10877.224} C_VEL
LIN {X 0,Y 404.325,Z 527.482,A -85,B 0,C 180,E1 -10878.723,E2 -10878.723} C_VEL
LIN {X 0,Y 403.707,Z 534.837,A -85,B 0,C 180,E1 -10880.227,E2 -10880.227} C_VEL
LIN {X 0,Y 403.249,Z 541.617,A -85,B 0,C 180,E1 -10881.985,E2 -10881.985} C_VEL
LIN {X 0,Y 402.938,Z 546.932,A -85,B 0,C 180,E1 -10883.821,E2 -10883.821} C_VEL
LIN {X 0,Y 402.931,Z 549.53,A -85,B 0,C 180,E1 -10884.996,E2 -10884.996} C_VEL
LIN {X 0,Y 402.827,Z 552.543,A -85,B 0,C 180,E1 -10886.999,E2 -10886.999} C_VEL
LIN {X 0,Y 402.907,Z 553.459,A -85,B 0,C 180,E1 -10888,E2 -10888} C_VEL
LIN {X 0,Y 402.865,Z 553.952,A -85,B 0,C 180,E1 -10889,E2 -10889} C_VEL
LIN {X 0,Y 402.871,Z 554.031,A -85,B 0,C 180,E1 -10889.999,E2 -10889.999} C_VEL
LIN {X 0,Y 402.911,Z 553.028,A -85,B 0,C 180,E1 -10891.998,E2 -10891.998} C_VEL
LIN {X 0,Y 402.858,Z 551.911,A -85,B 0,C 180,E1 -10892.999,E2 -10892.999} C_VEL
LIN {X 0,Y 402.857,Z 550.349,A -85,B 0,C 180,E1 -10894.001,E2 -10894.001} C_VEL
LIN {X 0,Y 402.915,Z 547.205,A -85,B 0,C 180,E1 -10895.504,E2 -10895.504} C_VEL
LIN {X 0,Y 403.074,Z 542.987,A -85,B 0,C 180,E1 -10897.01,E2 -10897.01} C_VEL
LIN {X 0,Y 403.371,Z 536.552,A -85,B 0,C 180,E1 -10898.768,E2 -10898.768} C_VEL
LIN {X 0,Y 403.76,Z 529.523,A -85,B 0,C 180,E1 -10900.277,E2 -10900.277} C_VEL
LIN {X 0,Y 404.406,Z 520.705,A -85,B 0,C 180,E1 -10901.782,E2 -10901.782} C_VEL
LIN {X 0,Y 405.057,Z 511.662,A -85,B 0,C 180,E1 -10903.035,E2 -10903.035} C_VEL
LIN {X 0,Y 405.735,Z 501.709,A -85,B 0,C 180,E1 -10904.161,E2 -10904.161} C_VEL
LIN {X 0,Y 406.448,Z 490.676,A -85,B 0,C 180,E1 -10905.16,E2 -10905.16} C_VEL
LIN {X 0,Y 407.258,Z 478.303,A -85,B 0,C 180,E1 -10906.027,E2 -10906.027} C_VEL
LIN {X 0,Y 407.861,Z 466.588,A -85,B 0,C 180,E1 -10906.646,E2 -10906.646} C_VEL
LIN {X 0,Y 408.42,Z 454.133,A -85,B 0,C 180,E1 -10907.105,E2 -10907.105} C_VEL
LIN {X 0,Y 408.712,Z 438.244,A -85,B 0,C 180,E1 -10907.447,E2 -10907.447} C_VEL
LIN {X 0,Y 409.365,Z 368.344,A -85,B 0,C 180,E1 -10908.679,E2 -10908.679} C_VEL
LIN {X 0,Y 405.465,Z 341.13,A -85,B 0,C 180,E1 -10909.359,E2 -10909.359} C_VEL
LIN {X 0,Y 406.393,Z 325.912,A -85,B 0,C 180,E1 -10912.361,E2 -10912.361} C_VEL
LIN {X 0,Y 407.044,Z 315.271,A -85,B 0,C 180,E1 -10914.479,E2 -10914.479} C_VEL
LIN {X 0,Y 405.08,Z 304.365,A -85,B 0,C 180,E1 -10916.813,E2 -10916.813} C_VEL
LIN {X 0,Y 404.249,Z 300.132,A -85,B 0,C 180,E1 -10917.758,E2 -10917.758} C_VEL
LIN {X 0,Y 404.136,Z 300.141,A -85,B 0,C 180,E1 -10921.557,E2 -10921.557} C_VEL
LIN {X 0,Y 404.182,Z 300.134,A -85,B 0,C 180,E1 -10925.015,E2 -10925.015} C_VEL
LIN {X 0,Y 404.146,Z 300.141,A -85,B 0,C 180,E1 -10928.756,E2 -10928.756} C_VEL
LIN {X 0,Y 404.118,Z 300.142,A -85,B 0,C 180,E1 -10931.599,E2 -10931.599} C_VEL
LIN {X 0,Y 404.141,Z 300.146,A -85,B 0,C 180,E1 -10934.521,E2 -10934.521} C_VEL
LIN {X 0,Y 404.134,Z 300.14,A -85,B 0,C 180,E1 -10937.295,E2 -10937.295} C_VEL
LIN {X 0,Y 404.163,Z 300.137,A -85,B 0,C 180,E1 -10939.954,E2 -10939.954} C_VEL
LIN {X 0,Y 404.133,Z 300.142,A -85,B 0,C 180,E1 -10943.123,E2 -10943.123} C_VEL
LIN {X 0,Y 404.138,Z 300.14,A -85,B 0,C 180,E1 -10946.187,E2 -10946.187} C_VEL
LIN {X 0,Y 404.149,Z 300.138,A -85,B 0,C 180,E1 -10949.715,E2 -10949.715} C_VEL
LIN {X 0,Y 404.188,Z 300.139,A -85,B 0,C 180,E1 -10953.122,E2 -10953.122} C_VEL
LIN {X 0,Y 404.169,Z 300.139,A -85,B 0,C 180,E1 -10955.334,E2 -10955.334} C_VEL
LIN {X 0,Y 404.13,Z 300.142,A -85,B 0,C 180,E1 -10958.58,E2 -10958.58} C_VEL
LIN {X 0,Y 404.201,Z 300.133,A -85,B 0,C 180,E1 -10961.762,E2 -10961.762} C_VEL
LIN {X 0,Y 404.198,Z 300.135,A -85,B 0,C 180,E1 -10964.882,E2 -10964.882} C_VEL
LIN {X 0,Y 404.248,Z 300.127,A -85,B 0,C 180,E1 -10967.958,E2 -10967.958} C_VEL
LIN {X 0,Y 404.424,Z 300.105,A -85,B 0,C 180,E1 -10972.1,E2 -10972.1} C_VEL
LIN {X 0,Y 404.414,Z 300.107,A -85,B 0,C 180,E1 -10974.015,E2 -10974.015} C_VEL
LIN {X 0,Y 404.472,Z 300.101,A -85,B 0,C 180,E1 -10978.009,E2 -10978.009} C_VEL
LIN {X 0,Y 404.601,Z 300.085,A -85,B 0,C 180,E1 -10980,E2 -10980} C_VEL
LIN {X 0,Y 404.414,Z 300.105,A -85,B 0,C 180,E1 -10982.989,E2 -10982.989} C_VEL
LIN {X 0,Y 404.359,Z 300.112,A -85,B 0,C 180,E1 -10986.988,E2 -10986.988} C_VEL
LIN {X 0,Y 404.249,Z 300.132,A -85,B 0,C 180,E1 -10990.012,E2 -10990.012} C_VEL
LIN {X 0,Y 404.257,Z 300.125,A -85,B 0,C 180,E1 -10993.212,E2 -10993.212} C_VEL
LIN {X 0,Y 404.21,Z 300.13,A -85,B 0,C 180,E1 -10997.009,E2 -10997.009} C_VEL
LIN {X 0,Y 404.155,Z 300.143,A -85,B 0,C 180,E1 -11000.352,E2 -11000.352} C_VEL
LIN {X 0,Y 404.152,Z 300.138,A -85,B 0,C 180,E1 -11003.576,E2 -11003.576} C_VEL
LIN {X 0,Y 404.173,Z 300.136,A -85,B 0,C 180,E1 -11005.767,E2 -11005.767} C_VEL
LIN {X 0,Y 404.187,Z 300.136,A -85,B 0,C 180,E1 -11008,E2 -11008} C_VEL
LIN {X 0,Y 404.131,Z 300.14,A -85,B 0,C 180,E1 -11011.559,E2 -11011.559} C_VEL
LIN {X 0,Y 404.178,Z 300.137,A -85,B 0,C 180,E1 -11015.017,E2 -11015.017} C_VEL
LIN {X 0,Y 404.128,Z 300.148,A -85,B 0,C 180,E1 -11018.76,E2 -11018.76} C_VEL
LIN {X 0,Y 404.107,Z 300.143,A -85,B 0,C 180,E1 -11021.599,E2 -11021.599} C_VEL
LIN {X 0,Y 404.139,Z 300.142,A -85,B 0,C 180,E1 -11024.523,E2 -11024.523} C_VEL
LIN {X 0,Y 404.119,Z 300.145,A -85,B 0,C 180,E1 -11027.295,E2 -11027.295} C_VEL
LIN {X 0,Y 404.128,Z 300.14,A -85,B 0,C 180,E1 -11029.952,E2 -11029.952} C_VEL
LIN {X 0,Y 404.131,Z 300.147,A -85,B 0,C 180,E1 -11033.127,E2 -11033.127} C_VEL
LIN {X 0,Y 404.141,Z 300.139,A -85,B 0,C 180,E1 -11036.189,E2 -11036.189} C_VEL
LIN {X 0,Y 404.14,Z 300.141,A -85,B 0,C 180,E1 -11039.716,E2 -11039.716} C_VEL
LIN {X 0,Y 404.101,Z 300.148,A -85,B 0,C 180,E1 -11043.117,E2 -11043.117} C_VEL
LIN {X 0,Y 404.147,Z 300.138,A -85,B 0,C 180,E1 -11046.425,E2 -11046.425} C_VEL
LIN {X 0,Y 404.191,Z 300.136,A -85,B 0,C 180,E1 -11049.875,E2 -11049.875} C_VEL
LIN {X 0,Y 404.216,Z 300.13,A -85,B 0,C 180,E1 -11052.994,E2 -11052.994} C_VEL
LIN {X 0,Y 404.284,Z 300.121,A -85,B 0,C 180,E1 -11056.94,E2 -11056.94} C_VEL
LIN {X 0,Y 404.24,Z 300.133,A -85,B 0,C 180,E1 -11059.989,E2 -11059.989} C_VEL
LIN {X 0,Y 404.345,Z 300.243,A -85,B 0,C 180,E1 -11061.782,E2 -11061.782} C_VEL
LIN {X 0,Y 405.795,Z 308.725,A -85,B 0,C 180,E1 -11063.787,E2 -11063.787} C_VEL
LIN {X 0,Y 405.739,Z 313.042,A -85,B 0,C 180,E1 -11064.752,E2 -11064.752} C_VEL
LIN {X 0,Y 409.836,Z 335.378,A -85,B 0,C 180,E1 -11065.333,E2 -11065.333} C_VEL
LIN {X 0,Y 408.725,Z 420.24,A -85,B 0,C 180,E1 -11066.84,E2 -11066.84} C_VEL
LIN {X 0,Y 408.291,Z 433.182,A -85,B 0,C 180,E1 -11067.257,E2 -11067.257} C_VEL
LIN {X 0,Y 407.826,Z 446.252,A -85,B 0,C 180,E1 -11067.893,E2 -11067.893} C_VEL
LIN {X 0,Y 407.224,Z 457.619,A -85,B 0,C 180,E1 -11068.641,E2 -11068.641} C_VEL
LIN {X 0,Y 406.513,Z 469.191,A -85,B 0,C 180,E1 -11069.629,E2 -11069.629} C_VEL
LIN {X 0,Y 405.763,Z 479.621,A -85,B 0,C 180,E1 -11070.745,E2 -11070.745} C_VEL
LIN {X 0,Y 405.52,Z 482.359,A -85,B 0,C 180,E1 -11071.083,E2 -11071.083} C_VEL
LIN {X 0,Y 404.568,Z 486.712,A -85,B 0,C 180,E1 -11071.64,E2 -11071.64} C_VEL
LIN {X 0,Y 401.227,Z 493.398,A -85,B 0,C 180,E1 -11072.573,E2 -11072.573} C_VEL
LIN {X 0,Y 397.919,Z 499.514,A -85,B 0,C 180,E1 -11073.586,E2 -11073.586} C_VEL
LIN {X 0,Y 397.022,Z 502.911,A -85,B 0,C 180,E1 -11074.262,E2 -11074.262} C_VEL
LIN {X 0,Y 396.571,Z 508.547,A -85,B 0,C 180,E1 -11075.594,E2 -11075.594} C_VEL
LIN {X 0,Y 396.299,Z 513.801,A -85,B 0,C 180,E1 -11077.132,E2 -11077.132} C_VEL
LIN {X 0,Y 396.041,Z 517.9,A -85,B 0,C 180,E1 -11078.676,E2 -11078.676} C_VEL
LIN {X 0,Y 395.81,Z 520.943,A -85,B 0,C 180,E1 -11080.228,E2 -11080.228} C_VEL
LIN {X 0,Y 395.768,Z 522.416,A -85,B 0,C 180,E1 -11081.265,E2 -11081.265} C_VEL
LIN {X 0,Y 395.722,Z 523.502,A -85,B 0,C 180,E1 -11082.366,E2 -11082.366} C_VEL
LIN {X 0,Y 395.651,Z 524.344,A -85,B 0,C 180,E1 -11084.4,E2 -11084.4} C_VEL
LIN {X 0,Y 395.719,Z 524.13,A -85,B 0,C 180,E1 -11085.451,E2 -11085.451} C_VEL
LIN {X 0,Y 395.745,Z 523.506,A -85,B 0,C 180,E1 -11086.508,E2 -11086.508} C_VEL
LIN {X 0,Y 395.796,Z 522.473,A -85,B 0,C 180,E1 -11087.57,E2 -11087.57} C_VEL
LIN {X 0,Y 395.932,Z 520.975,A -85,B 0,C 180,E1 -11088.634,E2 -11088.634} C_VEL
LIN {X 0,Y 396.218,Z 518.521,A -85,B 0,C 180,E1 -11089.931,E2 -11089.931} C_VEL
LIN {X 0,Y 396.496,Z 515.117,A -85,B 0,C 180,E1 -11091.308,E2 -11091.308} C_VEL
LIN {X 0,Y 397.021,Z 509.717,A -85,B 0,C 180,E1 -11093.001,E2 -11093.001} C_VEL
LIN {X 0,Y 397.657,Z 503.449,A -85,B 0,C 180,E1 -11094.54,E2 -11094.54} C_VEL
LIN {X 0,Y 398.506,Z 495.104,A -85,B 0,C 180,E1 -11096.162,E2 -11096.162} C_VEL
LIN {X 0,Y 399.326,Z 486.476,A -85,B 0,C 180,E1 -11097.516,E2 -11097.516} C_VEL
LIN {X 0,Y 400.272,Z 477.008,A -85,B 0,C 180,E1 -11098.724,E2 -11098.724} C_VEL
LIN {X 0,Y 401.218,Z 466.464,A -85,B 0,C 180,E1 -11099.804,E2 -11099.804} C_VEL
LIN {X 0,Y 402.113,Z 454.78,A -85,B 0,C 180,E1 -11100.751,E2 -11100.751} C_VEL
LIN {X 0,Y 402.829,Z 443.093,A -85,B 0,C 180,E1 -11101.481,E2 -11101.481} C_VEL
LIN {X 0,Y 403.401,Z 430.173,A -85,B 0,C 180,E1 -11102.061,E2 -11102.061} C_VEL
LIN {X 0,Y 403.77,Z 417.077,A -85,B 0,C 180,E1 -11102.434,E2 -11102.434} C_VEL
LIN {X 0,Y 405.097,Z 335.167,A -85,B 0,C 180,E1 -11103.919,E2 -11103.919} C_VEL
LIN {X 0,Y 400.534,Z 315.821,A -85,B 0,C 180,E1 -11104.575,E2 -11104.575} C_VEL
LIN {X 0,Y 399.799,Z 313.358,A -85,B 0,C 180,E1 -11104.692,E2 -11104.692} C_VEL
LIN {X 0,Y 397.089,Z 301.022,A -85,B 0,C 180,E1 -11107.79,E2 -11107.79} C_VEL
LIN {X 0,Y 397.091,Z 301.023,A -85,B 0,C 180,E1 -11110.909,E2 -11110.909} C_VEL
LIN {X 0,Y 397.103,Z 301.022,A -85,B 0,C 180,E1 -11113.648,E2 -11113.648} C_VEL
LIN {X 0,Y 397.104,Z 301.017,A -85,B 0,C 180,E1 -11116.521,E2 -11116.521} C_VEL
LIN {X 0,Y 397.116,Z 301.012,A -85,B 0,C 180,E1 -11120.423,E2 -11120.423} C_VEL
LIN {X 0,Y 397.109,Z 301.018,A -85,B 0,C 180,E1 -11124.265,E2 -11124.265} C_VEL
LIN {X 0,Y 397.116,Z 301.018,A -85,B 0,C 180,E1 -11126.727,E2 -11126.727} C_VEL
LIN {X 0,Y 397.126,Z 301.011,A -85,B 0,C 180,E1 -11130.296,E2 -11130.296} C_VEL
LIN {X 0,Y 397.195,Z 301.008,A -85,B 0,C 180,E1 -11132.61,E2 -11132.61} C_VEL
LIN {X 0,Y 397.134,Z 301.011,A -85,B 0,C 180,E1 -11135.982,E2 -11135.982} C_VEL
LIN {X 0,Y 397.14,Z 301.012,A -85,B 0,C 180,E1 -11139.705,E2 -11139.705} C_VEL
LIN {X 0,Y 397.183,Z 301.006,A -85,B 0,C 180,E1 -11142.845,E2 -11142.845} C_VEL
LIN {X 0,Y 397.229,Z 300.997,A -85,B 0,C 180,E1 -11146.703,E2 -11146.703} C_VEL
LIN {X 0,Y 397.218,Z 300.998,A -85,B 0,C 180,E1 -11149.809,E2 -11149.809} C_VEL
LIN {X 0,Y 397.363,Z 300.985,A -85,B 0,C 180,E1 -11152.888,E2 -11152.888} C_VEL
LIN {X 0,Y 397.253,Z 300.994,A -85,B 0,C 180,E1 -11154.925,E2 -11154.925} C_VEL
LIN {X 0,Y 397.449,Z 300.979,A -85,B 0,C 180,E1 -11157.973,E2 -11157.973} C_VEL
LIN {X 0,Y 397.579,Z 300.953,A -85,B 0,C 180,E1 -11160,E2 -11160} C_VEL
LIN {X 0,Y 397.376,Z 300.981,A -85,B 0,C 180,E1 -11163.041,E2 -11163.041} C_VEL
LIN {X 0,Y 397.362,Z 300.979,A -85,B 0,C 180,E1 -11167.112,E2 -11167.112} C_VEL
LIN {X 0,Y 397.217,Z 301.001,A -85,B 0,C 180,E1 -11170.191,E2 -11170.191} C_VEL
LIN {X 0,Y 397.227,Z 301,A -85,B 0,C 180,E1 -11173.321,E2 -11173.321} C_VEL
LIN {X 0,Y 397.183,Z 301.005,A -85,B 0,C 180,E1 -11177.155,E2 -11177.155} C_VEL
LIN {X 0,Y 397.103,Z 301.014,A -85,B 0,C 180,E1 -11180.73,E2 -11180.73} C_VEL
LIN {X 0,Y 397.13,Z 301.014,A -85,B 0,C 180,E1 -11184.018,E2 -11184.018} C_VEL
LIN {X 0,Y 397.195,Z 301.007,A -85,B 0,C 180,E1 -11187.39,E2 -11187.39} C_VEL
LIN {X 0,Y 397.079,Z 301.019,A -85,B 0,C 180,E1 -11190.882,E2 -11190.882} C_VEL
LIN {X 0,Y 397.125,Z 301.01,A -85,B 0,C 180,E1 -11194.493,E2 -11194.493} C_VEL
LIN {X 0,Y 397.102,Z 301.016,A -85,B 0,C 180,E1 -11198.275,E2 -11198.275} C_VEL
LIN {X 0,Y 397.09,Z 301.019,A -85,B 0,C 180,E1 -11200.909,E2 -11200.909} C_VEL
LIN {X 0,Y 397.102,Z 301.02,A -85,B 0,C 180,E1 -11203.648,E2 -11203.648} C_VEL
LIN {X 0,Y 397.104,Z 301.017,A -85,B 0,C 180,E1 -11206.521,E2 -11206.521} C_VEL
LIN {X 0,Y 397.114,Z 301.011,A -85,B 0,C 180,E1 -11210.423,E2 -11210.423} C_VEL
LIN {X 0,Y 397.11,Z 301.015,A -85,B 0,C 180,E1 -11214.265,E2 -11214.265} C_VEL
LIN {X 0,Y 397.117,Z 301.013,A -85,B 0,C 180,E1 -11216.727,E2 -11216.727} C_VEL
LIN {X 0,Y 397.172,Z 301.204,A -85,B 0,C 180,E1 -11220.736,E2 -11220.736} C_VEL
LIN {X 0,Y 399.661,Z 311.935,A -85,B 0,C 180,E1 -11223.309,E2 -11223.309} C_VEL
LIN {X 0,Y 401.053,Z 319.919,A -85,B 0,C 180,E1 -11225.129,E2 -11225.129} C_VEL
LIN {X 0,Y 399.69,Z 336.916,A -85,B 0,C 180,E1 -11228.633,E2 -11228.633} C_VEL
LIN {X 0,Y 399.443,Z 340.471,A -85,B 0,C 180,E1 -11229.359,E2 -11229.359} C_VEL
LIN {X 0,Y 403.999,Z 365.932,A -85,B 0,C 180,E1 -11230.132,E2 -11230.132} C_VEL
LIN {X 0,Y 404.633,Z 371.123,A -85,B 0,C 180,E1 -11230.268,E2 -11230.268} C_VEL
LIN {X 0,Y 403.415,Z 449.948,A -85,B 0,C 180,E1 -11231.724,E2 -11231.724} C_VEL
LIN {X 0,Y 402.804,Z 463.59,A -85,B 0,C 180,E1 -11232.188,E2 -11232.188} C_VEL
LIN {X 0,Y 401.964,Z 476.404,A -85,B 0,C 180,E1 -11232.839,E2 -11232.839} C_VEL
LIN {X 0,Y 400.945,Z 488.896,A -85,B 0,C 180,E1 -11233.712,E2 -11233.712} C_VEL
LIN {X 0,Y 399.941,Z 500.057,A -85,B 0,C 180,E1 -11234.716,E2 -11234.716} C_VEL
LIN {X 0,Y 399.028,Z 509.918,A -85,B 0,C 180,E1 -11235.826,E2 -11235.826} C_VEL
LIN {X 0,Y 398.14,Z 520.055,A -85,B 0,C 180,E1 -11237.252,E2 -11237.252} C_VEL
LIN {X 0,Y 397.172,Z 528.822,A -85,B 0,C 180,E1 -11238.775,E2 -11238.775} C_VEL
LIN {X 0,Y 396.607,Z 535.856,A -85,B 0,C 180,E1 -11240.308,E2 -11240.308} C_VEL
LIN {X 0,Y 396.197,Z 541.499,A -85,B 0,C 180,E1 -11241.841,E2 -11241.841} C_VEL
LIN {X 0,Y 395.929,Z 546.081,A -85,B 0,C 180,E1 -11243.425,E2 -11243.425} C_VEL
LIN {X 0,Y 395.843,Z 549.347,A -85,B 0,C 180,E1 -11244.906,E2 -11244.906} C_VEL
LIN {X 0,Y 395.776,Z 551.038,A -85,B 0,C 180,E1 -11245.926,E2 -11245.926} C_VEL
LIN {X 0,Y 395.803,Z 553.229,A -85,B 0,C 180,E1 -11247.964,E2 -11247.964} C_VEL
LIN {X 0,Y 395.795,Z 553.695,A -85,B 0,C 180,E1 -11248.982,E2 -11248.982} C_VEL
LIN {X 0,Y 395.797,Z 553.759,A -85,B 0,C 180,E1 -11249.999,E2 -11249.999} C_VEL
LIN {X 0,Y 395.81,Z 553.436,A -85,B 0,C 180,E1 -11251.017,E2 -11251.017} C_VEL
LIN {X 0,Y 395.825,Z 552.726,A -85,B 0,C 180,E1 -11252.034,E2 -11252.034} C_VEL
LIN {X 0,Y 395.759,Z 551.577,A -85,B 0,C 180,E1 -11253.053,E2 -11253.053} C_VEL
LIN {X 0,Y 395.78,Z 550,A -85,B 0,C 180,E1 -11254.072,E2 -11254.072} C_VEL
LIN {X 0,Y 395.827,Z 546.326,A -85,B 0,C 180,E1 -11255.805,E2 -11255.805} C_VEL
LIN {X 0,Y 396.057,Z 540.913,A -85,B 0,C 180,E1 -11257.647,E2 -11257.647} C_VEL
LIN {X 0,Y 396.433,Z 533.883,A -85,B 0,C 180,E1 -11259.437,E2 -11259.437} C_VEL
LIN {X 0,Y 396.887,Z 526.262,A -85,B 0,C 180,E1 -11260.973,E2 -11260.973} C_VEL
LIN {X 0,Y 397.562,Z 518.482,A -85,B 0,C 180,E1 -11262.246,E2 -11262.246} C_VEL
LIN {X 0,Y 398.256,Z 509.509,A -85,B 0,C 180,E1 -11263.456,E2 -11263.456} C_VEL
LIN {X 0,Y 398.988,Z 498.383,A -85,B 0,C 180,E1 -11264.667,E2 -11264.667} C_VEL
LIN {X 0,Y 399.778,Z 486.605,A -85,B 0,C 180,E1 -11265.68,E2 -11265.68} C_VEL
LIN {X 0,Y 400.581,Z 474.01,A -85,B 0,C 180,E1 -11266.498,E2 -11266.498} C_VEL
LIN {X 0,Y 401.209,Z 460.699,A -85,B 0,C 180,E1 -11267.127,E2 -11267.127} C_VEL
LIN {X 0,Y 401.681,Z 448.603,A -85,B 0,C 180,E1 -11267.5,E2 -11267.5} C_VEL
LIN {X 0,Y 402.561,Z 369.139,A -85,B 0,C 180,E1 -11268.936,E2 -11268.936} C_VEL
LIN {X 0,Y 398.533,Z 340.926,A -85,B 0,C 180,E1 -11269.642,E2 -11269.642} C_VEL
LIN {X 0,Y 399.508,Z 325.366,A -85,B 0,C 180,E1 -11272.768,E2 -11272.768} C_VEL
LIN {X 0,Y 400.04,Z 316.043,A -85,B 0,C 180,E1 -11274.661,E2 -11274.661} C_VEL
LIN {X 0,Y 398.013,Z 305.118,A -85,B 0,C 180,E1 -11277.044,E2 -11277.044} C_VEL
LIN {X 0,Y 397.2,Z 301.011,A -85,B 0,C 180,E1 -11278.007,E2 -11278.007} C_VEL
LIN {X 0,Y 397.079,Z 301.022,A -85,B 0,C 180,E1 -11281.836,E2 -11281.836} C_VEL
LIN {X 0,Y 397.123,Z 301.017,A -85,B 0,C 180,E1 -11284.492,E2 -11284.492} C_VEL
LIN {X 0,Y 397.096,Z 301.024,A -85,B 0,C 180,E1 -11288.274,E2 -11288.274} C_VEL
LIN {X 0,Y 397.084,Z 301.02,A -85,B 0,C 180,E1 -11290.908,E2 -11290.908} C_VEL
LIN {X 0,Y 397.096,Z 301.017,A -85,B 0,C 180,E1 -11293.647,E2 -11293.647} C_VEL
LIN {X 0,Y 397.099,Z 301.024,A -85,B 0,C 180,E1 -11296.52,E2 -11296.52} C_VEL
LIN {X 0,Y 397.109,Z 301.02,A -85,B 0,C 180,E1 -11300.422,E2 -11300.422} C_VEL
LIN {X 0,Y 397.102,Z 301.018,A -85,B 0,C 180,E1 -11304.265,E2 -11304.265} C_VEL
LIN {X 0,Y 397.108,Z 301.022,A -85,B 0,C 180,E1 -11306.726,E2 -11306.726} C_VEL
LIN {X 0,Y 397.127,Z 301.014,A -85,B 0,C 180,E1 -11310.296,E2 -11310.296} C_VEL
LIN {X 0,Y 397.187,Z 301.009,A -85,B 0,C 180,E1 -11312.609,E2 -11312.609} C_VEL
LIN {X 0,Y 397.124,Z 301.013,A -85,B 0,C 180,E1 -11315.981,E2 -11315.981} C_VEL
LIN {X 0,Y 397.13,Z 301.014,A -85,B 0,C 180,E1 -11319.704,E2 -11319.704} C_VEL
LIN {X 0,Y 397.173,Z 301.01,A -85,B 0,C 180,E1 -11322.844,E2 -11322.844} C_VEL
LIN {X 0,Y 397.219,Z 301.002,A -85,B 0,C 180,E1 -11326.702,E2 -11326.702} C_VEL
LIN {X 0,Y 397.21,Z 301.005,A -85,B 0,C 180,E1 -11329.809,E2 -11329.809} C_VEL
LIN {X 0,Y 397.354,Z 300.986,A -85,B 0,C 180,E1 -11332.888,E2 -11332.888} C_VEL
LIN {X 0,Y 397.245,Z 300.999,A -85,B 0,C 180,E1 -11334.925,E2 -11334.925} C_VEL
LIN {X 0,Y 397.441,Z 300.977,A -85,B 0,C 180,E1 -11337.973,E2 -11337.973} C_VEL
LIN {X 0,Y 397.571,Z 300.961,A -85,B 0,C 180,E1 -11340,E2 -11340} C_VEL
LIN {X 0,Y 397.372,Z 300.983,A -85,B 0,C 180,E1 -11343.042,E2 -11343.042} C_VEL
LIN {X 0,Y 397.308,Z 300.99,A -85,B 0,C 180,E1 -11347.113,E2 -11347.113} C_VEL
LIN {X 0,Y 397.208,Z 301.007,A -85,B 0,C 180,E1 -11350.191,E2 -11350.191} C_VEL
LIN {X 0,Y 397.218,Z 301.002,A -85,B 0,C 180,E1 -11353.321,E2 -11353.321} C_VEL
LIN {X 0,Y 397.162,Z 301.012,A -85,B 0,C 180,E1 -11356.447,E2 -11356.447} C_VEL
LIN {X 0,Y 397.139,Z 301.013,A -85,B 0,C 180,E1 -11359.648,E2 -11359.648} C_VEL
LIN {X 0,Y 397.103,Z 301.016,A -85,B 0,C 180,E1 -11363.033,E2 -11363.033} C_VEL
LIN {X 0,Y 397.125,Z 301.019,A -85,B 0,C 180,E1 -11366.259,E2 -11366.259} C_VEL
LIN {X 0,Y 397.114,Z 301.02,A -85,B 0,C 180,E1 -11368.544,E2 -11368.544} C_VEL
LIN {X 0,Y 397.071,Z 301.022,A -85,B 0,C 180,E1 -11372.072,E2 -11372.072} C_VEL
LIN {X 0,Y 397.112,Z 301.014,A -85,B 0,C 180,E1 -11375.504,E2 -11375.504} C_VEL
LIN {X 0,Y 397.086,Z 301.023,A -85,B 0,C 180,E1 -11378.856,E2 -11378.856} C_VEL
LIN {X 0,Y 397.055,Z 301.023,A -85,B 0,C 180,E1 -11382.269,E2 -11382.269} C_VEL
LIN {X 0,Y 397.081,Z 301.023,A -85,B 0,C 180,E1 -11385.07,E2 -11385.07} C_VEL
LIN {X 0,Y 397.049,Z 301.022,A -85,B 0,C 180,E1 -11388.024,E2 -11388.024} C_VEL
LIN {X 0,Y 397.089,Z 301.018,A -85,B 0,C 180,E1 -11391.725,E2 -11391.725} C_VEL
LIN {X 0,Y 397.121,Z 301.017,A -85,B 0,C 180,E1 -11395.508,E2 -11395.508} C_VEL
LIN {X 0,Y 397.075,Z 301.025,A -85,B 0,C 180,E1 -11399.119,E2 -11399.119} C_VEL
LIN {X 0,Y 397.059,Z 301.021,A -85,B 0,C 180,E1 -11402.253,E2 -11402.253} C_VEL
LIN {X 0,Y 397.101,Z 301.018,A -85,B 0,C 180,E1 -11404.866,E2 -11404.866} C_VEL
LIN {X 0,Y 397.094,Z 301.017,A -85,B 0,C 180,E1 -11408.182,E2 -11408.182} C_VEL
LIN {X 0,Y 397.157,Z 301.015,A -85,B 0,C 180,E1 -11411.427,E2 -11411.427} C_VEL
LIN {X 0,Y 397.177,Z 301.006,A -85,B 0,C 180,E1 -11414.609,E2 -11414.609} C_VEL
LIN {X 0,Y 397.212,Z 301.01,A -85,B 0,C 180,E1 -11417.743,E2 -11417.743} C_VEL
LIN {X 0,Y 397.281,Z 301.109,A -85,B 0,C 180,E1 -11421.577,E2 -11421.577} C_VEL
LIN {X 0,Y 398.8,Z 309.841,A -85,B 0,C 180,E1 -11423.677,E2 -11423.677} C_VEL
LIN {X 0,Y 398.824,Z 313.547,A -85,B 0,C 180,E1 -11424.471,E2 -11424.471} C_VEL
LIN {X 0,Y 403.021,Z 335.828,A -85,B 0,C 180,E1 -11425.061,E2 -11425.061} C_VEL
LIN {X 0,Y 401.877,Z 420.362,A -85,B 0,C 180,E1 -11426.586,E2 -11426.586} C_VEL
LIN {X 0,Y 401.457,Z 432.884,A -85,B 0,C 180,E1 -11426.99,E2 -11426.99} C_VEL
LIN {X 0,Y 400.939,Z 446.137,A -85,B 0,C 180,E1 -11427.637,E2 -11427.637} C_VEL
LIN {X 0,Y 400.359,Z 457.184,A -85,B 0,C 180,E1 -11428.366,E2 -11428.366} C_VEL
LIN {X 0,Y 399.619,Z 468.918,A -85,B 0,C 180,E1 -11429.371,E2 -11429.371} C_VEL
LIN {X 0,Y 398.844,Z 479.438,A -85,B 0,C 180,E1 -11430.506,E2 -11430.506} C_VEL
LIN {X 0,Y 398.074,Z 488.937,A -85,B 0,C 180,E1 -11431.771,E2 -11431.771} C_VEL
LIN {X 0,Y 397.349,Z 498.069,A -85,B 0,C 180,E1 -11433.296,E2 -11433.296} C_VEL
LIN {X 0,Y 397.022,Z 502.911,A -85,B 0,C 180,E1 -11434.262,E2 -11434.262} C_VEL
LIN {X 0,Y 396.146,Z 506.157,A -85,B 0,C 180,E1 -11434.964,E2 -11434.964} C_VEL
LIN {X 0,Y 392.948,Z 510.906,A -85,B 0,C 180,E1 -11436.141,E2 -11436.141} C_VEL
LIN {X 0,Y 389.805,Z 514.978,A -85,B 0,C 180,E1 -11437.39,E2 -11437.39} C_VEL
LIN {X 0,Y 389.032,Z 517.111,A -85,B 0,C 180,E1 -11438.194,E2 -11438.194} C_VEL
LIN {X 0,Y 388.844,Z 519.697,A -85,B 0,C 180,E1 -11439.362,E2 -11439.362} C_VEL
LIN {X 0,Y 388.714,Z 521.533,A -85,B 0,C 180,E1 -11440.417,E2 -11440.417} C_VEL
LIN {X 0,Y 388.628,Z 523.804,A -85,B 0,C 180,E1 -11442.433,E2 -11442.433} C_VEL
LIN {X 0,Y 388.567,Z 524.462,A -85,B 0,C 180,E1 -11443.6,E2 -11443.6} C_VEL
LIN {X 0,Y 388.563,Z 524.588,A -85,B 0,C 180,E1 -11444.669,E2 -11444.669} C_VEL
LIN {X 0,Y 388.653,Z 523.789,A -85,B 0,C 180,E1 -11446.584,E2 -11446.584} C_VEL
LIN {X 0,Y 388.758,Z 522.485,A -85,B 0,C 180,E1 -11447.899,E2 -11447.899} C_VEL
LIN {X 0,Y 389.066,Z 519.937,A -85,B 0,C 180,E1 -11449.523,E2 -11449.523} C_VEL
LIN {X 0,Y 389.396,Z 516.287,A -85,B 0,C 180,E1 -11451.16,E2 -11451.16} C_VEL
LIN {X 0,Y 389.871,Z 511.637,A -85,B 0,C 180,E1 -11452.738,E2 -11452.738} C_VEL
LIN {X 0,Y 390.566,Z 505.154,A -85,B 0,C 180,E1 -11454.449,E2 -11454.449} C_VEL
LIN {X 0,Y 391.446,Z 497.02,A -85,B 0,C 180,E1 -11456.142,E2 -11456.142} C_VEL
LIN {X 0,Y 392.306,Z 489.045,A -85,B 0,C 180,E1 -11457.471,E2 -11457.471} C_VEL
LIN {X 0,Y 393.248,Z 479.517,A -85,B 0,C 180,E1 -11458.768,E2 -11458.768} C_VEL
LIN {X 0,Y 394.309,Z 468.813,A -85,B 0,C 180,E1 -11459.938,E2 -11459.938} C_VEL
LIN {X 0,Y 395.27,Z 457.841,A -85,B 0,C 180,E1 -11460.891,E2 -11460.891} C_VEL
LIN {X 0,Y 395.985,Z 446.928,A -85,B 0,C 180,E1 -11461.635,E2 -11461.635} C_VEL
LIN {X 0,Y 396.623,Z 433.725,A -85,B 0,C 180,E1 -11462.301,E2 -11462.301} C_VEL
LIN {X 0,Y 397.103,Z 420.968,A -85,B 0,C 180,E1 -11462.727,E2 -11462.727} C_VEL
LIN {X 0,Y 398.608,Z 336.399,A -85,B 0,C 180,E1 -11464.297,E2 -11464.297} C_VEL
LIN {X 0,Y 394.235,Z 317.94,A -85,B 0,C 180,E1 -11464.943,E2 -11464.943} C_VEL
LIN {X 0,Y 392.657,Z 313.696,A -85,B 0,C 180,E1 -11465.145,E2 -11465.145} C_VEL
LIN {X 0,Y 390.072,Z 301.897,A -85,B 0,C 180,E1 -11468.186,E2 -11468.186} C_VEL
LIN {X 0,Y 390.033,Z 301.901,A -85,B 0,C 180,E1 -11471.813,E2 -11471.813} C_VEL
LIN {X 0,Y 390.046,Z 301.901,A -85,B 0,C 180,E1 -11475.354,E2 -11475.354} C_VEL
LIN {X 0,Y 390.033,Z 301.903,A -85,B 0,C 180,E1 -11478.187,E2 -11478.187} C_VEL
LIN {X 0,Y 390.093,Z 301.886,A -85,B 0,C 180,E1 -11480.908,E2 -11480.908} C_VEL
LIN {X 0,Y 390.086,Z 301.895,A -85,B 0,C 180,E1 -11484.793,E2 -11484.793} C_VEL
LIN {X 0,Y 390.025,Z 301.901,A -85,B 0,C 180,E1 -11488.496,E2 -11488.496} C_VEL
LIN {X 0,Y 390.119,Z 301.887,A -85,B 0,C 180,E1 -11492.07,E2 -11492.07} C_VEL
LIN {X 0,Y 390.081,Z 301.893,A -85,B 0,C 180,E1 -11495.519,E2 -11495.519} C_VEL
LIN {X 0,Y 390.057,Z 301.896,A -85,B 0,C 180,E1 -11498.878,E2 -11498.878} C_VEL
LIN {X 0,Y 390.129,Z 301.884,A -85,B 0,C 180,E1 -11502.167,E2 -11502.167} C_VEL
LIN {X 0,Y 390.145,Z 301.881,A -85,B 0,C 180,E1 -11505.393,E2 -11505.393} C_VEL
LIN {X 0,Y 390.148,Z 301.883,A -85,B 0,C 180,E1 -11508.571,E2 -11508.571} C_VEL
LIN {X 0,Y 390.344,Z 301.862,A -85,B 0,C 180,E1 -11511.994,E2 -11511.994} C_VEL
LIN {X 0,Y 390.225,Z 301.869,A -85,B 0,C 180,E1 -11514.833,E2 -11514.833} C_VEL
LIN {X 0,Y 390.418,Z 301.854,A -85,B 0,C 180,E1 -11517.937,E2 -11517.937} C_VEL
LIN {X 0,Y 390.548,Z 301.829,A -85,B 0,C 180,E1 -11520,E2 -11520} C_VEL
LIN {X 0,Y 390.31,Z 301.861,A -85,B 0,C 180,E1 -11523.096,E2 -11523.096} C_VEL
LIN {X 0,Y 390.327,Z 301.855,A -85,B 0,C 180,E1 -11526.202,E2 -11526.202} C_VEL
LIN {X 0,Y 390.315,Z 301.866,A -85,B 0,C 180,E1 -11528.282,E2 -11528.282} C_VEL
LIN {X 0,Y 390.171,Z 301.879,A -85,B 0,C 180,E1 -11532.483,E2 -11532.483} C_VEL
LIN {X 0,Y 390.14,Z 301.879,A -85,B 0,C 180,E1 -11535.677,E2 -11535.677} C_VEL
LIN {X 0,Y 390.106,Z 301.89,A -85,B 0,C 180,E1 -11538.922,E2 -11538.922} C_VEL
LIN {X 0,Y 390.038,Z 301.894,A -85,B 0,C 180,E1 -11542.234,E2 -11542.234} C_VEL
LIN {X 0,Y 390.12,Z 301.879,A -85,B 0,C 180,E1 -11545.743,E2 -11545.743} C_VEL
LIN {X 0,Y 390.06,Z 301.892,A -85,B 0,C 180,E1 -11549.11,E2 -11549.11} C_VEL
LIN {X 0,Y 390.043,Z 301.9,A -85,B 0,C 180,E1 -11552.722,E2 -11552.722} C_VEL
LIN {X 0,Y 390.056,Z 301.895,A -85,B 0,C 180,E1 -11555.825,E2 -11555.825} C_VEL
LIN {X 0,Y 390.07,Z 301.899,A -85,B 0,C 180,E1 -11559.218,E2 -11559.218} C_VEL
LIN {X 0,Y 390.044,Z 301.898,A -85,B 0,C 180,E1 -11562.374,E2 -11562.374} C_VEL
LIN {X 0,Y 390.046,Z 301.9,A -85,B 0,C 180,E1 -11565.354,E2 -11565.354} C_VEL
LIN {X 0,Y 390.032,Z 301.9,A -85,B 0,C 180,E1 -11568.187,E2 -11568.187} C_VEL
LIN {X 0,Y 390.089,Z 301.885,A -85,B 0,C 180,E1 -11570.907,E2 -11570.907} C_VEL
LIN {X 0,Y 390.087,Z 301.892,A -85,B 0,C 180,E1 -11574.793,E2 -11574.793} C_VEL
LIN {X 0,Y 390.026,Z 301.899,A -85,B 0,C 180,E1 -11578.495,E2 -11578.495} C_VEL
LIN {X 0,Y 390.098,Z 301.925,A -85,B 0,C 180,E1 -11580.301,E2 -11580.301} C_VEL
LIN {X 0,Y 393.016,Z 314.576,A -85,B 0,C 180,E1 -11583.395,E2 -11583.395} C_VEL
LIN {X 0,Y 394.162,Z 321.082,A -85,B 0,C 180,E1 -11584.909,E2 -11584.909} C_VEL
LIN {X 0,Y 392.855,Z 337.281,A -85,B 0,C 180,E1 -11588.314,E2 -11588.314} C_VEL
LIN {X 0,Y 392.634,Z 340.106,A -85,B 0,C 180,E1 -11588.902,E2 -11588.902} C_VEL
LIN {X 0,Y 396.922,Z 363.294,A -85,B 0,C 180,E1 -11589.652,E2 -11589.652} C_VEL
LIN {X 0,Y 398.076,Z 372.138,A -85,B 0,C 180,E1 -11589.895,E2 -11589.895} C_VEL
LIN {X 0,Y 396.809,Z 449.513,A -85,B 0,C 180,E1 -11591.347,E2 -11591.347} C_VEL
LIN {X 0,Y 396.191,Z 463.087,A -85,B 0,C 180,E1 -11591.814,E2 -11591.814} C_VEL
LIN {X 0,Y 395.297,Z 475.982,A -85,B 0,C 180,E1 -11592.474,E2 -11592.474} C_VEL
LIN {X 0,Y 394.307,Z 487.719,A -85,B 0,C 180,E1 -11593.297,E2 -11593.297} C_VEL
LIN {X 0,Y 393.199,Z 499.047,A -85,B 0,C 180,E1 -11594.315,E2 -11594.315} C_VEL
LIN {X 0,Y 392.186,Z 509.286,A -85,B 0,C 180,E1 -11595.47,E2 -11595.47} C_VEL
LIN {X 0,Y 391.37,Z 518.503,A -85,B 0,C 180,E1 -11596.764,E2 -11596.764} C_VEL
LIN {X 0,Y 390.379,Z 527.484,A -85,B 0,C 180,E1 -11598.314,E2 -11598.314} C_VEL
LIN {X 0,Y 389.668,Z 534.739,A -85,B 0,C 180,E1 -11599.871,E2 -11599.871} C_VEL
LIN {X 0,Y 389.136,Z 541.392,A -85,B 0,C 180,E1 -11601.692,E2 -11601.692} C_VEL
LIN {X 0,Y 388.852,Z 545.809,A -85,B 0,C 180,E1 -11603.253,E2 -11603.253} C_VEL
LIN {X 0,Y 388.739,Z 549.163,A -85,B 0,C 180,E1 -11604.813,E2 -11604.813} C_VEL
LIN {X 0,Y 388.7,Z 550.84,A -85,B 0,C 180,E1 -11605.852,E2 -11605.852} C_VEL
LIN {X 0,Y 388.7,Z 552.995,A -85,B 0,C 180,E1 -11607.927,E2 -11607.927} C_VEL
LIN {X 0,Y 388.725,Z 553.438,A -85,B 0,C 180,E1 -11608.963,E2 -11608.963} C_VEL
LIN {X 0,Y 388.725,Z 553.487,A -85,B 0,C 180,E1 -11609.999,E2 -11609.999} C_VEL
LIN {X 0,Y 388.74,Z 553.15,A -85,B 0,C 180,E1 -11611.035,E2 -11611.035} C_VEL
LIN {X 0,Y 388.724,Z 552.42,A -85,B 0,C 180,E1 -11612.071,E2 -11612.071} C_VEL
LIN {X 0,Y 388.664,Z 551.243,A -85,B 0,C 180,E1 -11613.109,E2 -11613.109} C_VEL
LIN {X 0,Y 388.72,Z 548.712,A -85,B 0,C 180,E1 -11614.666,E2 -11614.666} C_VEL
LIN {X 0,Y 388.794,Z 545.155,A -85,B 0,C 180,E1 -11616.226,E2 -11616.226} C_VEL
LIN {X 0,Y 388.986,Z 540.476,A -85,B 0,C 180,E1 -11617.787,E2 -11617.787} C_VEL
LIN {X 0,Y 389.384,Z 533.403,A -85,B 0,C 180,E1 -11619.61,E2 -11619.61} C_VEL
LIN {X 0,Y 389.878,Z 525.731,A -85,B 0,C 180,E1 -11621.173,E2 -11621.173} C_VEL
LIN {X 0,Y 390.557,Z 517.878,A -85,B 0,C 180,E1 -11622.47,E2 -11622.47} C_VEL
LIN {X 0,Y 391.391,Z 507.689,A -85,B 0,C 180,E1 -11623.834,E2 -11623.834} C_VEL
LIN {X 0,Y 392.086,Z 497.586,A -85,B 0,C 180,E1 -11624.931,E2 -11624.931} C_VEL
LIN {X 0,Y 392.878,Z 485.618,A -85,B 0,C 180,E1 -11625.963,E2 -11625.963} C_VEL
LIN {X 0,Y 393.733,Z 472.786,A -85,B 0,C 180,E1 -11626.794,E2 -11626.794} C_VEL
LIN {X 0,Y 394.369,Z 459.886,A -85,B 0,C 180,E1 -11627.4,E2 -11627.4} C_VEL
LIN {X 0,Y 394.847,Z 447.278,A -85,B 0,C 180,E1 -11627.779,E2 -11627.779} C_VEL
LIN {X 0,Y 395.754,Z 370.034,A -85,B 0,C 180,E1 -11629.195,E2 -11629.195} C_VEL
LIN {X 0,Y 391.558,Z 340.7,A -85,B 0,C 180,E1 -11629.938,E2 -11629.938} C_VEL
LIN {X 0,Y 392.536,Z 326.128,A -85,B 0,C 180,E1 -11632.917,E2 -11632.917} C_VEL
LIN {X 0,Y 393.113,Z 318.142,A -85,B 0,C 180,E1 -11634.56,E2 -11634.56} C_VEL
LIN {X 0,Y 391.492,Z 308.6,A -85,B 0,C 180,E1 -11636.665,E2 -11636.665} C_VEL
LIN {X 0,Y 390.175,Z 301.886,A -85,B 0,C 180,E1 -11638.225,E2 -11638.225} C_VEL
LIN {X 0,Y 390.029,Z 301.904,A -85,B 0,C 180,E1 -11642.124,E2 -11642.124} C_VEL
LIN {X 0,Y 390.082,Z 301.89,A -85,B 0,C 180,E1 -11645.206,E2 -11645.206} C_VEL
LIN {X 0,Y 390.063,Z 301.893,A -85,B 0,C 180,E1 -11649.217,E2 -11649.217} C_VEL
LIN {X 0,Y 390.038,Z 301.903,A -85,B 0,C 180,E1 -11652.373,E2 -11652.373} C_VEL
LIN {X 0,Y 390.041,Z 301.895,A -85,B 0,C 180,E1 -11655.354,E2 -11655.354} C_VEL
LIN {X 0,Y 390.027,Z 301.9,A -85,B 0,C 180,E1 -11658.186,E2 -11658.186} C_VEL
LIN {X 0,Y 390.086,Z 301.894,A -85,B 0,C 180,E1 -11660.907,E2 -11660.907} C_VEL
LIN {X 0,Y 390.079,Z 301.898,A -85,B 0,C 180,E1 -11664.792,E2 -11664.792} C_VEL
LIN {X 0,Y 390.042,Z 301.899,A -85,B 0,C 180,E1 -11668.497,E2 -11668.497} C_VEL
LIN {X 0,Y 390.109,Z 301.887,A -85,B 0,C 180,E1 -11672.069,E2 -11672.069} C_VEL
LIN {X 0,Y 390.072,Z 301.893,A -85,B 0,C 180,E1 -11675.519,E2 -11675.519} C_VEL
LIN {X 0,Y 390.047,Z 301.899,A -85,B 0,C 180,E1 -11678.877,E2 -11678.877} C_VEL
LIN {X 0,Y 390.119,Z 301.886,A -85,B 0,C 180,E1 -11682.166,E2 -11682.166} C_VEL
LIN {X 0,Y 390.135,Z 301.89,A -85,B 0,C 180,E1 -11685.392,E2 -11685.392} C_VEL
LIN {X 0,Y 390.14,Z 301.883,A -85,B 0,C 180,E1 -11688.571,E2 -11688.571} C_VEL
LIN {X 0,Y 390.335,Z 301.86,A -85,B 0,C 180,E1 -11691.993,E2 -11691.993} C_VEL
LIN {X 0,Y 390.217,Z 301.874,A -85,B 0,C 180,E1 -11694.833,E2 -11694.833} C_VEL
LIN {X 0,Y 390.41,Z 301.853,A -85,B 0,C 180,E1 -11697.937,E2 -11697.937} C_VEL
LIN {X 0,Y 390.54,Z 301.837,A -85,B 0,C 180,E1 -11700,E2 -11700} C_VEL
LIN {X 0,Y 390.306,Z 301.863,A -85,B 0,C 180,E1 -11703.097,E2 -11703.097} C_VEL
LIN {X 0,Y 390.266,Z 301.868,A -85,B 0,C 180,E1 -11706.506,E2 -11706.506} C_VEL
LIN {X 0,Y 390.194,Z 301.877,A -85,B 0,C 180,E1 -11709.329,E2 -11709.329} C_VEL
LIN {X 0,Y 390.185,Z 301.879,A -85,B 0,C 180,E1 -11713.439,E2 -11713.439} C_VEL
LIN {X 0,Y 390.141,Z 301.883,A -85,B 0,C 180,E1 -11717.309,E2 -11717.309} C_VEL
LIN {X 0,Y 390.079,Z 301.895,A -85,B 0,C 180,E1 -11720.471,E2 -11720.471} C_VEL
LIN {X 0,Y 390.067,Z 301.898,A -85,B 0,C 180,E1 -11724.482,E2 -11724.482} C_VEL
LIN {X 0,Y 390.11,Z 301.889,A -85,B 0,C 180,E1 -11727.931,E2 -11727.931} C_VEL
LIN {X 0,Y 390.016,Z 301.898,A -85,B 0,C 180,E1 -11731.505,E2 -11731.505} C_VEL
LIN {X 0,Y 390.078,Z 301.892,A -85,B 0,C 180,E1 -11735.208,E2 -11735.208} C_VEL
LIN {X 0,Y 390.051,Z 301.897,A -85,B 0,C 180,E1 -11739.097,E2 -11739.097} C_VEL
LIN {X 0,Y 390.03,Z 301.899,A -85,B 0,C 180,E1 -11742.374,E2 -11742.374} C_VEL
LIN {X 0,Y 390.038,Z 301.898,A -85,B 0,C 180,E1 -11745.355,E2 -11745.355} C_VEL
LIN {X 0,Y 390.012,Z 301.899,A -85,B 0,C 180,E1 -11748.186,E2 -11748.186} C_VEL
LIN {X 0,Y 390.055,Z 301.899,A -85,B 0,C 180,E1 -11750.905,E2 -11750.905} C_VEL
LIN {X 0,Y 390.081,Z 301.894,A -85,B 0,C 180,E1 -11754.794,E2 -11754.794} C_VEL
LIN {X 0,Y 390.02,Z 301.898,A -85,B 0,C 180,E1 -11758.497,E2 -11758.497} C_VEL
LIN {X 0,Y 390.013,Z 301.9,A -85,B 0,C 180,E1 -11762.004,E2 -11762.004} C_VEL
LIN {X 0,Y 390.041,Z 301.902,A -85,B 0,C 180,E1 -11765.518,E2 -11765.518} C_VEL
LIN {X 0,Y 390.055,Z 301.895,A -85,B 0,C 180,E1 -11768.879,E2 -11768.879} C_VEL
LIN {X 0,Y 390.111,Z 301.888,A -85,B 0,C 180,E1 -11772.167,E2 -11772.167} C_VEL
LIN {X 0,Y 390.143,Z 301.887,A -85,B 0,C 180,E1 -11775.394,E2 -11775.394} C_VEL
LIN {X 0,Y 390.132,Z 301.884,A -85,B 0,C 180,E1 -11778.572,E2 -11778.572} C_VEL
LIN {X 0,Y 390.245,Z 302.066,A -85,B 0,C 180,E1 -11781.391,E2 -11781.391} C_VEL
LIN {X 0,Y 391.807,Z 310.964,A -85,B 0,C 180,E1 -11783.564,E2 -11783.564} C_VEL
LIN {X 0,Y 391.834,Z 313.534,A -85,B 0,C 180,E1 -11784.16,E2 -11784.16} C_VEL
LIN {X 0,Y 396.188,Z 337.091,A -85,B 0,C 180,E1 -11784.797,E2 -11784.797} C_VEL
LIN {X 0,Y 395.019,Z 420.756,A -85,B 0,C 180,E1 -11786.334,E2 -11786.334} C_VEL
LIN {X 0,Y 394.577,Z 433.209,A -85,B 0,C 180,E1 -11786.744,E2 -11786.744} C_VEL
LIN {X 0,Y 394.089,Z 445.567,A -85,B 0,C 180,E1 -11787.352,E2 -11787.352} C_VEL
LIN {X 0,Y 393.487,Z 456.638,A -85,B 0,C 180,E1 -11788.082,E2 -11788.082} C_VEL
LIN {X 0,Y 392.818,Z 467.271,A -85,B 0,C 180,E1 -11788.976,E2 -11788.976} C_VEL
LIN {X 0,Y 392.026,Z 478.138,A -85,B 0,C 180,E1 -11790.129,E2 -11790.129} C_VEL
LIN {X 0,Y 391.217,Z 487.03,A -85,B 0,C 180,E1 -11791.287,E2 -11791.287} C_VEL
LIN {X 0,Y 390.454,Z 496.658,A -85,B 0,C 180,E1 -11792.838,E2 -11792.838} C_VEL
LIN {X 0,Y 389.876,Z 504.322,A -85,B 0,C 180,E1 -11794.395,E2 -11794.395} C_VEL
LIN {X 0,Y 389.49,Z 509.577,A -85,B 0,C 180,E1 -11795.696,E2 -11795.696} C_VEL
LIN {X 0,Y 389.189,Z 514.66,A -85,B 0,C 180,E1 -11797.263,E2 -11797.263} C_VEL
LIN {X 0,Y 389.032,Z 517.111,A -85,B 0,C 180,E1 -11798.194,E2 -11798.194} C_VEL
LIN {X 0,Y 388.291,Z 519.026,A -85,B 0,C 180,E1 -11799.01,E2 -11799.01} C_VEL
LIN {X 0,Y 385.309,Z 521.582,A -85,B 0,C 180,E1 -11800.356,E2 -11800.356} C_VEL
LIN {X 0,Y 382.78,Z 523.108,A -85,B 0,C 180,E1 -11801.463,E2 -11801.463} C_VEL
LIN {X 0,Y 381.647,Z 523.974,A -85,B 0,C 180,E1 -11802.328,E2 -11802.328} C_VEL
LIN {X 0,Y 381.529,Z 524.194,A -85,B 0,C 180,E1 -11802.623,E2 -11802.623} C_VEL
LIN {X 0,Y 381.479,Z 524.773,A -85,B 0,C 180,E1 -11803.858,E2 -11803.858} C_VEL
LIN {X 0,Y 381.474,Z 524.825,A -85,B 0,C 180,E1 -11804.948,E2 -11804.948} C_VEL
LIN {X 0,Y 381.583,Z 524.034,A -85,B 0,C 180,E1 -11806.716,E2 -11806.716} C_VEL
LIN {X 0,Y 381.72,Z 522.464,A -85,B 0,C 180,E1 -11808.24,E2 -11808.24} C_VEL
LIN {X 0,Y 382.142,Z 518.999,A -85,B 0,C 180,E1 -11810.29,E2 -11810.29} C_VEL
LIN {X 0,Y 382.612,Z 514.468,A -85,B 0,C 180,E1 -11812.121,E2 -11812.121} C_VEL
LIN {X 0,Y 383.201,Z 508.972,A -85,B 0,C 180,E1 -11813.797,E2 -11813.797} C_VEL
LIN {X 0,Y 384.013,Z 501.986,A -85,B 0,C 180,E1 -11815.473,E2 -11815.473} C_VEL
LIN {X 0,Y 384.888,Z 494.525,A -85,B 0,C 180,E1 -11816.916,E2 -11816.916} C_VEL
LIN {X 0,Y 385.811,Z 485.984,A -85,B 0,C 180,E1 -11818.27,E2 -11818.27} C_VEL
LIN {X 0,Y 386.877,Z 476.192,A -85,B 0,C 180,E1 -11819.522,E2 -11819.522} C_VEL
LIN {X 0,Y 387.964,Z 465.394,A -85,B 0,C 180,E1 -11820.63,E2 -11820.63} C_VEL
LIN {X 0,Y 388.928,Z 453.397,A -85,B 0,C 180,E1 -11821.604,E2 -11821.604} C_VEL
LIN {X 0,Y 389.713,Z 441.341,A -85,B 0,C 180,E1 -11822.336,E2 -11822.336} C_VEL
LIN {X 0,Y 390.295,Z 428.581,A -85,B 0,C 180,E1 -11822.89,E2 -11822.89} C_VEL
LIN {X 0,Y 390.667,Z 415.738,A -85,B 0,C 180,E1 -11823.239,E2 -11823.239} C_VEL
LIN {X 0,Y 392.034,Z 337.226,A -85,B 0,C 180,E1 -11824.706,E2 -11824.706} C_VEL
LIN {X 0,Y 387.877,Z 319.759,A -85,B 0,C 180,E1 -11825.336,E2 -11825.336} C_VEL
LIN {X 0,Y 385.511,Z 313.94,A -85,B 0,C 180,E1 -11825.639,E2 -11825.639} C_VEL
LIN {X 0,Y 383.026,Z 302.771,A -85,B 0,C 180,E1 -11828.598,E2 -11828.598} C_VEL
LIN {X 0,Y 382.986,Z 302.779,A -85,B 0,C 180,E1 -11831.347,E2 -11831.347} C_VEL
LIN {X 0,Y 382.998,Z 302.78,A -85,B 0,C 180,E1 -11834.303,E2 -11834.303} C_VEL
LIN {X 0,Y 383.012,Z 302.774,A -85,B 0,C 180,E1 -11837.24,E2 -11837.24} C_VEL
LIN {X 0,Y 383.018,Z 302.767,A -85,B 0,C 180,E1 -11840.413,E2 -11840.413} C_VEL
LIN {X 0,Y 383.027,Z 302.772,A -85,B 0,C 180,E1 -11844.044,E2 -11844.044} C_VEL
LIN {X 0,Y 382.988,Z 302.777,A -85,B 0,C 180,E1 -11847.578,E2 -11847.578} C_VEL
LIN {X 0,Y 382.993,Z 302.771,A -85,B 0,C 180,E1 -11850.3,E2 -11850.3} C_VEL
LIN {X 0,Y 383.058,Z 302.769,A -85,B 0,C 180,E1 -11852.698,E2 -11852.698} C_VEL
LIN {X 0,Y 383.054,Z 302.772,A -85,B 0,C 180,E1 -11855.04,E2 -11855.04} C_VEL
LIN {X 0,Y 382.994,Z 302.774,A -85,B 0,C 180,E1 -11858.469,E2 -11858.469} C_VEL
LIN {X 0,Y 383.09,Z 302.762,A -85,B 0,C 180,E1 -11861.828,E2 -11861.828} C_VEL
LIN {X 0,Y 383.111,Z 302.758,A -85,B 0,C 180,E1 -11865.118,E2 -11865.118} C_VEL
LIN {X 0,Y 383.097,Z 302.762,A -85,B 0,C 180,E1 -11868.358,E2 -11868.358} C_VEL
LIN {X 0,Y 383.304,Z 302.738,A -85,B 0,C 180,E1 -11871.933,E2 -11871.933} C_VEL
LIN {X 0,Y 383.197,Z 302.745,A -85,B 0,C 180,E1 -11874.738,E2 -11874.738} C_VEL
LIN {X 0,Y 383.385,Z 302.729,A -85,B 0,C 180,E1 -11877.899,E2 -11877.899} C_VEL
LIN {X 0,Y 383.518,Z 302.704,A -85,B 0,C 180,E1 -11880,E2 -11880} C_VEL
LIN {X 0,Y 383.247,Z 302.741,A -85,B 0,C 180,E1 -11883.154,E2 -11883.154} C_VEL
LIN {X 0,Y 383.285,Z 302.732,A -85,B 0,C 180,E1 -11886.316,E2 -11886.316} C_VEL
LIN {X 0,Y 383.261,Z 302.744,A -85,B 0,C 180,E1 -11888.436,E2 -11888.436} C_VEL
LIN {X 0,Y 383.137,Z 302.758,A -85,B 0,C 180,E1 -11892.716,E2 -11892.716} C_VEL
LIN {X 0,Y 383.081,Z 302.759,A -85,B 0,C 180,E1 -11895.973,E2 -11895.973} C_VEL
LIN {X 0,Y 383.061,Z 302.766,A -85,B 0,C 180,E1 -11899.284,E2 -11899.284} C_VEL
LIN {X 0,Y 382.996,Z 302.776,A -85,B 0,C 180,E1 -11902.666,E2 -11902.666} C_VEL
LIN {X 0,Y 383.081,Z 302.756,A -85,B 0,C 180,E1 -11906.123,E2 -11906.123} C_VEL
LIN {X 0,Y 383.041,Z 302.772,A -85,B 0,C 180,E1 -11908.493,E2 -11908.493} C_VEL
LIN {X 0,Y 383.01,Z 302.773,A -85,B 0,C 180,E1 -11912.15,E2 -11912.15} C_VEL
LIN {X 0,Y 383.019,Z 302.768,A -85,B 0,C 180,E1 -11914.668,E2 -11914.668} C_VEL
LIN {X 0,Y 383,Z 302.774,A -85,B 0,C 180,E1 -11917.903,E2 -11917.903} C_VEL
LIN {X 0,Y 382.985,Z 302.779,A -85,B 0,C 180,E1 -11921.347,E2 -11921.347} C_VEL
LIN {X 0,Y 382.997,Z 302.776,A -85,B 0,C 180,E1 -11924.303,E2 -11924.303} C_VEL
LIN {X 0,Y 383.012,Z 302.778,A -85,B 0,C 180,E1 -11927.24,E2 -11927.24} C_VEL
LIN {X 0,Y 383.015,Z 302.767,A -85,B 0,C 180,E1 -11930.414,E2 -11930.414} C_VEL
LIN {X 0,Y 383.027,Z 302.769,A -85,B 0,C 180,E1 -11934.044,E2 -11934.044} C_VEL
LIN {X 0,Y 382.99,Z 302.777,A -85,B 0,C 180,E1 -11937.578,E2 -11937.578} C_VEL
LIN {X 0,Y 383.026,Z 302.845,A -85,B 0,C 180,E1 -11939.889,E2 -11939.889} C_VEL
LIN {X 0,Y 385.863,Z 314.871,A -85,B 0,C 180,E1 -11942.913,E2 -11942.913} C_VEL
LIN {X 0,Y 387.304,Z 322.606,A -85,B 0,C 180,E1 -11944.759,E2 -11944.759} C_VEL
LIN {X 0,Y 385.99,Z 337.67,A -85,B 0,C 180,E1 -11947.984,E2 -11947.984} C_VEL
LIN {X 0,Y 385.847,Z 340.189,A -85,B 0,C 180,E1 -11948.469,E2 -11948.469} C_VEL
LIN {X 0,Y 390.071,Z 362.123,A -85,B 0,C 180,E1 -11949.192,E2 -11949.192} C_VEL
LIN {X 0,Y 391.564,Z 373.337,A -85,B 0,C 180,E1 -11949.511,E2 -11949.511} C_VEL
LIN {X 0,Y 390.242,Z 449.099,A -85,B 0,C 180,E1 -11950.955,E2 -11950.955} C_VEL
LIN {X 0,Y 389.573,Z 462.675,A -85,B 0,C 180,E1 -11951.426,E2 -11951.426} C_VEL
LIN {X 0,Y 388.625,Z 475.608,A -85,B 0,C 180,E1 -11952.095,E2 -11952.095} C_VEL
LIN {X 0,Y 387.535,Z 488.142,A -85,B 0,C 180,E1 -11952.996,E2 -11952.996} C_VEL
LIN {X 0,Y 386.384,Z 499.333,A -85,B 0,C 180,E1 -11954.031,E2 -11954.031} C_VEL
LIN {X 0,Y 385.301,Z 509.445,A -85,B 0,C 180,E1 -11955.204,E2 -11955.204} C_VEL
LIN {X 0,Y 384.454,Z 518.579,A -85,B 0,C 180,E1 -11956.521,E2 -11956.521} C_VEL
LIN {X 0,Y 383.392,Z 527.503,A -85,B 0,C 180,E1 -11958.098,E2 -11958.098} C_VEL
LIN {X 0,Y 382.664,Z 534.707,A -85,B 0,C 180,E1 -11959.684,E2 -11959.684} C_VEL
LIN {X 0,Y 382.092,Z 541.295,A -85,B 0,C 180,E1 -11961.538,E2 -11961.538} C_VEL
LIN {X 0,Y 381.785,Z 545.673,A -85,B 0,C 180,E1 -11963.127,E2 -11963.127} C_VEL
LIN {X 0,Y 381.644,Z 548.991,A -85,B 0,C 180,E1 -11964.716,E2 -11964.716} C_VEL
LIN {X 0,Y 381.625,Z 550.651,A -85,B 0,C 180,E1 -11965.775,E2 -11965.775} C_VEL
LIN {X 0,Y 381.549,Z 551.908,A -85,B 0,C 180,E1 -11966.832,E2 -11966.832} C_VEL
LIN {X 0,Y 381.598,Z 552.759,A -85,B 0,C 180,E1 -11967.888,E2 -11967.888} C_VEL
LIN {X 0,Y 381.639,Z 553.18,A -85,B 0,C 180,E1 -11968.944,E2 -11968.944} C_VEL
LIN {X 0,Y 381.656,Z 553.214,A -85,B 0,C 180,E1 -11969.999,E2 -11969.999} C_VEL
LIN {X 0,Y 381.672,Z 552.861,A -85,B 0,C 180,E1 -11971.054,E2 -11971.054} C_VEL
LIN {X 0,Y 381.624,Z 552.106,A -85,B 0,C 180,E1 -11972.11,E2 -11972.11} C_VEL
LIN {X 0,Y 381.631,Z 549.295,A -85,B 0,C 180,E1 -11974.224,E2 -11974.224} C_VEL
LIN {X 0,Y 381.688,Z 545.316,A -85,B 0,C 180,E1 -11976.119,E2 -11976.119} C_VEL
LIN {X 0,Y 381.908,Z 540.018,A -85,B 0,C 180,E1 -11977.932,E2 -11977.932} C_VEL
LIN {X 0,Y 382.262,Z 534.026,A -85,B 0,C 180,E1 -11979.523,E2 -11979.523} C_VEL
LIN {X 0,Y 382.748,Z 526.543,A -85,B 0,C 180,E1 -11981.115,E2 -11981.115} C_VEL
LIN {X 0,Y 383.453,Z 518.921,A -85,B 0,C 180,E1 -11982.435,E2 -11982.435} C_VEL
LIN {X 0,Y 384.233,Z 509.675,A -85,B 0,C 180,E1 -11983.755,E2 -11983.755} C_VEL
LIN {X 0,Y 384.957,Z 499.364,A -85,B 0,C 180,E1 -11984.943,E2 -11984.943} C_VEL
LIN {X 0,Y 385.767,Z 487.918,A -85,B 0,C 180,E1 -11985.994,E2 -11985.994} C_VEL
LIN {X 0,Y 386.61,Z 476.033,A -85,B 0,C 180,E1 -11986.84,E2 -11986.84} C_VEL
LIN {X 0,Y 387.29,Z 463.668,A -85,B 0,C 180,E1 -11987.49,E2 -11987.49} C_VEL
LIN {X 0,Y 387.905,Z 449.944,A -85,B 0,C 180,E1 -11987.972,E2 -11987.972} C_VEL
LIN {X 0,Y 388.72,Z 398.113,A -85,B 0,C 180,E1 -11988.957,E2 -11988.957} C_VEL
LIN {X 0,Y 388.903,Z 370.664,A -85,B 0,C 180,E1 -11989.471,E2 -11989.471} C_VEL
LIN {X 0,Y 384.59,Z 340.505,A -85,B 0,C 180,E1 -11990.237,E2 -11990.237} C_VEL
LIN {X 0,Y 385.672,Z 325.546,A -85,B 0,C 180,E1 -11993.349,E2 -11993.349} C_VEL
LIN {X 0,Y 386.112,Z 318.887,A -85,B 0,C 180,E1 -11994.748,E2 -11994.748} C_VEL
LIN {X 0,Y 384.138,Z 307.961,A -85,B 0,C 180,E1 -11997.217,E2 -11997.217} C_VEL
LIN {X 0,Y 383.104,Z 302.767,A -85,B 0,C 180,E1 -11998.45,E2 -11998.45} C_VEL
LIN {X 0,Y 382.984,Z 302.778,A -85,B 0,C 180,E1 -12002.421,E2 -12002.421} C_VEL
LIN {X 0,Y 383.022,Z 302.774,A -85,B 0,C 180,E1 -12005.954,E2 -12005.954} C_VEL
LIN {X 0,Y 383.009,Z 302.772,A -85,B 0,C 180,E1 -12009.585,E2 -12009.585} C_VEL
LIN {X 0,Y 383,Z 302.776,A -85,B 0,C 180,E1 -12012.778,E2 -12012.778} C_VEL
LIN {X 0,Y 382.994,Z 302.774,A -85,B 0,C 180,E1 -12015.789,E2 -12015.789} C_VEL
LIN {X 0,Y 382.984,Z 302.779,A -85,B 0,C 180,E1 -12018.795,E2 -12018.795} C_VEL
LIN {X 0,Y 382.995,Z 302.774,A -85,B 0,C 180,E1 -12022.095,E2 -12022.095} C_VEL
LIN {X 0,Y 383.011,Z 302.772,A -85,B 0,C 180,E1 -12025.331,E2 -12025.331} C_VEL
LIN {X 0,Y 383.03,Z 302.769,A -85,B 0,C 180,E1 -12027.852,E2 -12027.852} C_VEL
LIN {X 0,Y 383.056,Z 302.766,A -85,B 0,C 180,E1 -12031.72,E2 -12031.72} C_VEL
LIN {X 0,Y 383.044,Z 302.774,A -85,B 0,C 180,E1 -12035.039,E2 -12035.039} C_VEL
LIN {X 0,Y 382.984,Z 302.775,A -85,B 0,C 180,E1 -12038.468,E2 -12038.468} C_VEL
LIN {X 0,Y 383.054,Z 302.767,A -85,B 0,C 180,E1 -12041.826,E2 -12041.826} C_VEL
LIN {X 0,Y 383.101,Z 302.765,A -85,B 0,C 180,E1 -12045.118,E2 -12045.118} C_VEL
LIN {X 0,Y 383.089,Z 302.761,A -85,B 0,C 180,E1 -12048.358,E2 -12048.358} C_VEL
LIN {X 0,Y 383.295,Z 302.738,A -85,B 0,C 180,E1 -12051.933,E2 -12051.933} C_VEL
LIN {X 0,Y 383.189,Z 302.749,A -85,B 0,C 180,E1 -12054.738,E2 -12054.738} C_VEL
LIN {X 0,Y 383.378,Z 302.729,A -85,B 0,C 180,E1 -12057.899,E2 -12057.899} C_VEL
LIN {X 0,Y 383.51,Z 302.712,A -85,B 0,C 180,E1 -12060,E2 -12060} C_VEL
LIN {X 0,Y 383.243,Z 302.743,A -85,B 0,C 180,E1 -12063.154,E2 -12063.154} C_VEL
LIN {X 0,Y 383.23,Z 302.745,A -85,B 0,C 180,E1 -12066.494,E2 -12066.494} C_VEL
LIN {X 0,Y 383.141,Z 302.757,A -85,B 0,C 180,E1 -12069.502,E2 -12069.502} C_VEL
LIN {X 0,Y 383.116,Z 302.76,A -85,B 0,C 180,E1 -12073.537,E2 -12073.537} C_VEL
LIN {X 0,Y 383.087,Z 302.762,A -85,B 0,C 180,E1 -12077.456,E2 -12077.456} C_VEL
LIN {X 0,Y 383.02,Z 302.772,A -85,B 0,C 180,E1 -12080.647,E2 -12080.647} C_VEL
LIN {X 0,Y 383.013,Z 302.773,A -85,B 0,C 180,E1 -12083.809,E2 -12083.809} C_VEL
LIN {X 0,Y 383.071,Z 302.768,A -85,B 0,C 180,E1 -12086.124,E2 -12086.124} C_VEL
LIN {X 0,Y 383.032,Z 302.775,A -85,B 0,C 180,E1 -12088.494,E2 -12088.494} C_VEL
LIN {X 0,Y 383.002,Z 302.775,A -85,B 0,C 180,E1 -12092.151,E2 -12092.151} C_VEL
LIN {X 0,Y 383.011,Z 302.778,A -85,B 0,C 180,E1 -12094.669,E2 -12094.669} C_VEL
LIN {X 0,Y 382.987,Z 302.774,A -85,B 0,C 180,E1 -12097.903,E2 -12097.903} C_VEL
LIN {X 0,Y 382.956,Z 302.779,A -85,B 0,C 180,E1 -12101.351,E2 -12101.351} C_VEL
LIN {X 0,Y 382.99,Z 302.775,A -85,B 0,C 180,E1 -12104.304,E2 -12104.304} C_VEL
LIN {X 0,Y 383.006,Z 302.775,A -85,B 0,C 180,E1 -12107.241,E2 -12107.241} C_VEL
LIN {X 0,Y 382.982,Z 302.776,A -85,B 0,C 180,E1 -12110.42,E2 -12110.42} C_VEL
LIN {X 0,Y 383.02,Z 302.77,A -85,B 0,C 180,E1 -12114.045,E2 -12114.045} C_VEL
LIN {X 0,Y 382.983,Z 302.777,A -85,B 0,C 180,E1 -12117.579,E2 -12117.579} C_VEL
LIN {X 0,Y 382.973,Z 302.776,A -85,B 0,C 180,E1 -12120.3,E2 -12120.3} C_VEL
LIN {X 0,Y 383.001,Z 302.773,A -85,B 0,C 180,E1 -12124.046,E2 -12124.046} C_VEL
LIN {X 0,Y 382.989,Z 302.78,A -85,B 0,C 180,E1 -12127.335,E2 -12127.335} C_VEL
LIN {X 0,Y 383.058,Z 302.765,A -85,B 0,C 180,E1 -12130.717,E2 -12130.717} C_VEL
LIN {X 0,Y 383.08,Z 302.765,A -85,B 0,C 180,E1 -12134.028,E2 -12134.028} C_VEL
LIN {X 0,Y 383.133,Z 302.758,A -85,B 0,C 180,E1 -12137.285,E2 -12137.285} C_VEL
LIN {X 0,Y 383.213,Z 302.879,A -85,B 0,C 180,E1 -12141.166,E2 -12141.166} C_VEL
LIN {X 0,Y 384.815,Z 312.091,A -85,B 0,C 180,E1 -12143.446,E2 -12143.446} C_VEL
LIN {X 0,Y 384.91,Z 313.743,A -85,B 0,C 180,E1 -12143.841,E2 -12143.841} C_VEL
LIN {X 0,Y 389.38,Z 337.134,A -85,B 0,C 180,E1 -12144.501,E2 -12144.501} C_VEL
LIN {X 0,Y 388.09,Z 421.892,A -85,B 0,C 180,E1 -12146.092,E2 -12146.092} C_VEL
LIN {X 0,Y 387.681,Z 434.873,A -85,B 0,C 180,E1 -12146.547,E2 -12146.547} C_VEL
LIN {X 0,Y 387.147,Z 447.447,A -85,B 0,C 180,E1 -12147.199,E2 -12147.199} C_VEL
LIN {X 0,Y 386.416,Z 459.439,A -85,B 0,C 180,E1 -12148.047,E2 -12148.047} C_VEL
LIN {X 0,Y 385.637,Z 470.827,A -85,B 0,C 180,E1 -12149.087,E2 -12149.087} C_VEL
LIN {X 0,Y 384.818,Z 481.115,A -85,B 0,C 180,E1 -12150.262,E2 -12150.262} C_VEL
LIN {X 0,Y 384.005,Z 490.364,A -85,B 0,C 180,E1 -12151.574,E2 -12151.574} C_VEL
LIN {X 0,Y 383.233,Z 499.338,A -85,B 0,C 180,E1 -12153.155,E2 -12153.155} C_VEL
LIN {X 0,Y 382.66,Z 506.569,A -85,B 0,C 180,E1 -12154.741,E2 -12154.741} C_VEL
LIN {X 0,Y 382.301,Z 512.339,A -85,B 0,C 180,E1 -12156.333,E2 -12156.333} C_VEL
LIN {X 0,Y 381.945,Z 517.417,A -85,B 0,C 180,E1 -12158.156,E2 -12158.156} C_VEL
LIN {X 0,Y 381.729,Z 520.359,A -85,B 0,C 180,E1 -12159.538,E2 -12159.538} C_VEL
LIN {X 0,Y 381.626,Z 522.081,A -85,B 0,C 180,E1 -12160.613,E2 -12160.613} C_VEL
LIN {X 0,Y 381.529,Z 524.194,A -85,B 0,C 180,E1 -12162.623,E2 -12162.623} C_VEL
LIN {X 0,Y 380.784,Z 524.73,A -85,B 0,C 180,E1 -12163.5,E2 -12163.5} C_VEL
LIN {X 0,Y 377.901,Z 525.013,A -85,B 0,C 180,E1 -12164.932,E2 -12164.932} C_VEL
LIN {X 0,Y 375.543,Z 524.714,A -85,B 0,C 180,E1 -12166.089,E2 -12166.089} C_VEL
LIN {X 0,Y 374.581,Z 524.184,A -85,B 0,C 180,E1 -12166.981,E2 -12166.981} C_VEL
LIN {X 0,Y 374.528,Z 523.914,A -85,B 0,C 180,E1 -12167.281,E2 -12167.281} C_VEL
LIN {X 0,Y 374.703,Z 522.443,A -85,B 0,C 180,E1 -12168.594,E2 -12168.594} C_VEL
LIN {X 0,Y 375.093,Z 519.257,A -85,B 0,C 180,E1 -12170.473,E2 -12170.473} C_VEL
LIN {X 0,Y 375.503,Z 515.683,A -85,B 0,C 180,E1 -12171.983,E2 -12171.983} C_VEL
LIN {X 0,Y 376.116,Z 510.432,A -85,B 0,C 180,E1 -12173.708,E2 -12173.708} C_VEL
LIN {X 0,Y 376.907,Z 503.853,A -85,B 0,C 180,E1 -12175.396,E2 -12175.396} C_VEL
LIN {X 0,Y 377.978,Z 495.242,A -85,B 0,C 180,E1 -12177.136,E2 -12177.136} C_VEL
LIN {X 0,Y 378.96,Z 486.717,A -85,B 0,C 180,E1 -12178.526,E2 -12178.526} C_VEL
LIN {X 0,Y 380.079,Z 477.245,A -85,B 0,C 180,E1 -12179.777,E2 -12179.777} C_VEL
LIN {X 0,Y 381.229,Z 466.41,A -85,B 0,C 180,E1 -12180.923,E2 -12180.923} C_VEL
LIN {X 0,Y 382.227,Z 454.599,A -85,B 0,C 180,E1 -12181.913,E2 -12181.913} C_VEL
LIN {X 0,Y 383.093,Z 442.247,A -85,B 0,C 180,E1 -12182.693,E2 -12182.693} C_VEL
LIN {X 0,Y 383.718,Z 429.308,A -85,B 0,C 180,E1 -12183.272,E2 -12183.272} C_VEL
LIN {X 0,Y 384.13,Z 415.99,A -85,B 0,C 180,E1 -12183.644,E2 -12183.644} C_VEL
LIN {X 0,Y 385.623,Z 338.57,A -85,B 0,C 180,E1 -12185.11,E2 -12185.11} C_VEL
LIN {X 0,Y 381.817,Z 322.658,A -85,B 0,C 180,E1 -12185.702,E2 -12185.702} C_VEL
LIN {X 0,Y 378.361,Z 314.224,A -85,B 0,C 180,E1 -12186.152,E2 -12186.152} C_VEL
LIN {X 0,Y 375.972,Z 303.649,A -85,B 0,C 180,E1 -12189,E2 -12189} C_VEL
LIN {X 0,Y 375.934,Z 303.66,A -85,B 0,C 180,E1 -12192.3,E2 -12192.3} C_VEL
LIN {X 0,Y 375.929,Z 303.66,A -85,B 0,C 180,E1 -12195.269,E2 -12195.269} C_VEL
LIN {X 0,Y 375.937,Z 303.662,A -85,B 0,C 180,E1 -12198.399,E2 -12198.399} C_VEL
LIN {X 0,Y 375.976,Z 303.648,A -85,B 0,C 180,E1 -12201.729,E2 -12201.729} C_VEL
LIN {X 0,Y 375.981,Z 303.652,A -85,B 0,C 180,E1 -12205.333,E2 -12205.333} C_VEL
LIN {X 0,Y 375.959,Z 303.653,A -85,B 0,C 180,E1 -12208.438,E2 -12208.438} C_VEL
LIN {X 0,Y 375.997,Z 303.647,A -85,B 0,C 180,E1 -12212.141,E2 -12212.141} C_VEL
LIN {X 0,Y 376.007,Z 303.645,A -85,B 0,C 180,E1 -12214.539,E2 -12214.539} C_VEL
LIN {X 0,Y 375.964,Z 303.65,A -85,B 0,C 180,E1 -12218.046,E2 -12218.046} C_VEL
LIN {X 0,Y 376.025,Z 303.64,A -85,B 0,C 180,E1 -12221.474,E2 -12221.474} C_VEL
LIN {X 0,Y 376.059,Z 303.637,A -85,B 0,C 180,E1 -12224.832,E2 -12224.832} C_VEL
LIN {X 0,Y 376.05,Z 303.641,A -85,B 0,C 180,E1 -12228.136,E2 -12228.136} C_VEL
LIN {X 0,Y 376.258,Z 303.614,A -85,B 0,C 180,E1 -12231.878,E2 -12231.878} C_VEL
LIN {X 0,Y 376.17,Z 303.62,A -85,B 0,C 180,E1 -12234.64,E2 -12234.64} C_VEL
LIN {X 0,Y 376.352,Z 303.605,A -85,B 0,C 180,E1 -12237.86,E2 -12237.86} C_VEL
LIN {X 0,Y 376.487,Z 303.58,A -85,B 0,C 180,E1 -12240,E2 -12240} C_VEL
LIN {X 0,Y 376.185,Z 303.621,A -85,B 0,C 180,E1 -12243.213,E2 -12243.213} C_VEL
LIN {X 0,Y 376.245,Z 303.609,A -85,B 0,C 180,E1 -12246.435,E2 -12246.435} C_VEL
LIN {X 0,Y 376.206,Z 303.621,A -85,B 0,C 180,E1 -12248.595,E2 -12248.595} C_VEL
LIN {X 0,Y 376.049,Z 303.63,A -85,B 0,C 180,E1 -12251.863,E2 -12251.863} C_VEL
LIN {X 0,Y 376.059,Z 303.633,A -85,B 0,C 180,E1 -12255.167,E2 -12255.167} C_VEL
LIN {X 0,Y 376.025,Z 303.647,A -85,B 0,C 180,E1 -12258.526,E2 -12258.526} C_VEL
LIN {X 0,Y 375.959,Z 303.646,A -85,B 0,C 180,E1 -12261.955,E2 -12261.955} C_VEL
LIN {X 0,Y 376.006,Z 303.637,A -85,B 0,C 180,E1 -12265.461,E2 -12265.461} C_VEL
LIN {X 0,Y 375.971,Z 303.647,A -85,B 0,C 180,E1 -12269.079,E2 -12269.079} C_VEL
LIN {X 0,Y 375.95,Z 303.654,A -85,B 0,C 180,E1 -12272.829,E2 -12272.829} C_VEL
LIN {X 0,Y 375.958,Z 303.655,A -85,B 0,C 180,E1 -12275.416,E2 -12275.416} C_VEL
LIN {X 0,Y 375.974,Z 303.648,A -85,B 0,C 180,E1 -12278.27,E2 -12278.27} C_VEL
LIN {X 0,Y 375.936,Z 303.659,A -85,B 0,C 180,E1 -12281.601,E2 -12281.601} C_VEL
LIN {X 0,Y 375.928,Z 303.659,A -85,B 0,C 180,E1 -12285.269,E2 -12285.269} C_VEL
LIN {X 0,Y 375.936,Z 303.655,A -85,B 0,C 180,E1 -12288.399,E2 -12288.399} C_VEL
LIN {X 0,Y 375.974,Z 303.648,A -85,B 0,C 180,E1 -12291.73,E2 -12291.73} C_VEL
LIN {X 0,Y 375.982,Z 303.652,A -85,B 0,C 180,E1 -12295.333,E2 -12295.333} C_VEL
LIN {X 0,Y 375.961,Z 303.652,A -85,B 0,C 180,E1 -12298.438,E2 -12298.438} C_VEL
LIN {X 0,Y 375.993,Z 303.836,A -85,B 0,C 180,E1 -12299.481,E2 -12299.481} C_VEL
LIN {X 0,Y 378.669,Z 314.95,A -85,B 0,C 180,E1 -12302.354,E2 -12302.354} C_VEL
LIN {X 0,Y 380.42,Z 323.963,A -85,B 0,C 180,E1 -12304.562,E2 -12304.562} C_VEL
LIN {X 0,Y 379.58,Z 334.3,A -85,B 0,C 180,E1 -12306.83,E2 -12306.83} C_VEL
LIN {X 0,Y 379.044,Z 339.669,A -85,B 0,C 180,E1 -12307.983,E2 -12307.983} C_VEL
LIN {X 0,Y 383.487,Z 362.414,A -85,B 0,C 180,E1 -12308.761,E2 -12308.761} C_VEL
LIN {X 0,Y 385.052,Z 372.995,A -85,B 0,C 180,E1 -12309.08,E2 -12309.08} C_VEL
LIN {X 0,Y 383.697,Z 448.6,A -85,B 0,C 180,E1 -12310.545,E2 -12310.545} C_VEL
LIN {X 0,Y 382.971,Z 462.32,A -85,B 0,C 180,E1 -12311.024,E2 -12311.024} C_VEL
LIN {X 0,Y 381.971,Z 475.282,A -85,B 0,C 180,E1 -12311.703,E2 -12311.703} C_VEL
LIN {X 0,Y 380.941,Z 487.039,A -85,B 0,C 180,E1 -12312.554,E2 -12312.554} C_VEL
LIN {X 0,Y 379.722,Z 498.383,A -85,B 0,C 180,E1 -12313.605,E2 -12313.605} C_VEL
LIN {X 0,Y 378.578,Z 508.637,A -85,B 0,C 180,E1 -12314.798,E2 -12314.798} C_VEL
LIN {X 0,Y 377.545,Z 518.682,A -85,B 0,C 180,E1 -12316.27,E2 -12316.27} C_VEL
LIN {X 0,Y 376.432,Z 527.536,A -85,B 0,C 180,E1 -12317.875,E2 -12317.875} C_VEL
LIN {X 0,Y 375.672,Z 534.672,A -85,B 0,C 180,E1 -12319.49,E2 -12319.49} C_VEL
LIN {X 0,Y 375.037,Z 541.199,A -85,B 0,C 180,E1 -12321.377,E2 -12321.377} C_VEL
LIN {X 0,Y 374.726,Z 545.537,A -85,B 0,C 180,E1 -12322.997,E2 -12322.997} C_VEL
LIN {X 0,Y 374.555,Z 548.819,A -85,B 0,C 180,E1 -12324.616,E2 -12324.616} C_VEL
LIN {X 0,Y 374.551,Z 550.462,A -85,B 0,C 180,E1 -12325.695,E2 -12325.695} C_VEL
LIN {X 0,Y 374.463,Z 551.702,A -85,B 0,C 180,E1 -12326.772,E2 -12326.772} C_VEL
LIN {X 0,Y 374.496,Z 552.519,A -85,B 0,C 180,E1 -12327.848,E2 -12327.848} C_VEL
LIN {X 0,Y 374.555,Z 552.924,A -85,B 0,C 180,E1 -12328.924,E2 -12328.924} C_VEL
LIN {X 0,Y 374.588,Z 552.941,A -85,B 0,C 180,E1 -12329.999,E2 -12329.999} C_VEL
LIN {X 0,Y 374.586,Z 552.571,A -85,B 0,C 180,E1 -12331.074,E2 -12331.074} C_VEL
LIN {X 0,Y 374.524,Z 551.784,A -85,B 0,C 180,E1 -12332.15,E2 -12332.15} C_VEL
LIN {X 0,Y 374.559,Z 548.935,A -85,B 0,C 180,E1 -12334.303,E2 -12334.303} C_VEL
LIN {X 0,Y 374.586,Z 545.299,A -85,B 0,C 180,E1 -12336.071,E2 -12336.071} C_VEL
LIN {X 0,Y 374.765,Z 541.272,A -85,B 0,C 180,E1 -12337.542,E2 -12337.542} C_VEL
LIN {X 0,Y 375.075,Z 535.689,A -85,B 0,C 180,E1 -12339.164,E2 -12339.164} C_VEL
LIN {X 0,Y 375.524,Z 528.704,A -85,B 0,C 180,E1 -12340.786,E2 -12340.786} C_VEL
LIN {X 0,Y 376.332,Z 519.948,A -85,B 0,C 180,E1 -12342.401,E2 -12342.401} C_VEL
LIN {X 0,Y 377.123,Z 510.96,A -85,B 0,C 180,E1 -12343.744,E2 -12343.744} C_VEL
LIN {X 0,Y 377.793,Z 501.569,A -85,B 0,C 180,E1 -12344.898,E2 -12344.898} C_VEL
LIN {X 0,Y 378.632,Z 490.152,A -85,B 0,C 180,E1 -12346.027,E2 -12346.027} C_VEL
LIN {X 0,Y 379.553,Z 477.899,A -85,B 0,C 180,E1 -12346.955,E2 -12346.955} C_VEL
LIN {X 0,Y 380.335,Z 465.058,A -85,B 0,C 180,E1 -12347.681,E2 -12347.681} C_VEL
LIN {X 0,Y 380.987,Z 452.235,A -85,B 0,C 180,E1 -12348.171,E2 -12348.171} C_VEL
LIN {X 0,Y 381.367,Z 434.151,A -85,B 0,C 180,E1 -12348.567,E2 -12348.567} C_VEL
LIN {X 0,Y 382.034,Z 371.042,A -85,B 0,C 180,E1 -12349.759,E2 -12349.759} C_VEL
LIN {X 0,Y 377.674,Z 340.134,A -85,B 0,C 180,E1 -12350.579,E2 -12350.579} C_VEL
LIN {X 0,Y 378.834,Z 324.969,A -85,B 0,C 180,E1 -12353.796,E2 -12353.796} C_VEL
LIN {X 0,Y 379.1,Z 319.77,A -85,B 0,C 180,E1 -12354.914,E2 -12354.914} C_VEL
LIN {X 0,Y 376.796,Z 307.288,A -85,B 0,C 180,E1 -12357.793,E2 -12357.793} C_VEL
LIN {X 0,Y 376.04,Z 303.647,A -85,B 0,C 180,E1 -12358.686,E2 -12358.686} C_VEL
LIN {X 0,Y 375.947,Z 303.652,A -85,B 0,C 180,E1 -12362.729,E2 -12362.729} C_VEL
LIN {X 0,Y 375.954,Z 303.65,A -85,B 0,C 180,E1 -12365.414,E2 -12365.414} C_VEL
LIN {X 0,Y 375.968,Z 303.655,A -85,B 0,C 180,E1 -12368.269,E2 -12368.269} C_VEL
LIN {X 0,Y 375.929,Z 303.654,A -85,B 0,C 180,E1 -12371.6,E2 -12371.6} C_VEL
LIN {X 0,Y 375.923,Z 303.654,A -85,B 0,C 180,E1 -12375.267,E2 -12375.267} C_VEL
LIN {X 0,Y 375.93,Z 303.658,A -85,B 0,C 180,E1 -12378.398,E2 -12378.398} C_VEL
LIN {X 0,Y 375.97,Z 303.648,A -85,B 0,C 180,E1 -12381.728,E2 -12381.728} C_VEL
LIN {X 0,Y 375.973,Z 303.649,A -85,B 0,C 180,E1 -12385.332,E2 -12385.332} C_VEL
LIN {X 0,Y 375.97,Z 303.651,A -85,B 0,C 180,E1 -12388.439,E2 -12388.439} C_VEL
LIN {X 0,Y 375.995,Z 303.645,A -85,B 0,C 180,E1 -12392.141,E2 -12392.141} C_VEL
LIN {X 0,Y 375.998,Z 303.647,A -85,B 0,C 180,E1 -12394.538,E2 -12394.538} C_VEL
LIN {X 0,Y 375.955,Z 303.65,A -85,B 0,C 180,E1 -12398.045,E2 -12398.045} C_VEL
LIN {X 0,Y 376,Z 303.648,A -85,B 0,C 180,E1 -12401.473,E2 -12401.473} C_VEL
LIN {X 0,Y 376.049,Z 303.641,A -85,B 0,C 180,E1 -12404.832,E2 -12404.832} C_VEL
LIN {X 0,Y 376.041,Z 303.64,A -85,B 0,C 180,E1 -12408.136,E2 -12408.136} C_VEL
LIN {X 0,Y 376.248,Z 303.616,A -85,B 0,C 180,E1 -12411.877,E2 -12411.877} C_VEL
LIN {X 0,Y 376.162,Z 303.624,A -85,B 0,C 180,E1 -12414.64,E2 -12414.64} C_VEL
LIN {X 0,Y 376.344,Z 303.606,A -85,B 0,C 180,E1 -12417.86,E2 -12417.86} C_VEL
LIN {X 0,Y 376.479,Z 303.588,A -85,B 0,C 180,E1 -12420,E2 -12420} C_VEL
LIN {X 0,Y 376.18,Z 303.624,A -85,B 0,C 180,E1 -12423.213,E2 -12423.213} C_VEL
LIN {X 0,Y 376.199,Z 303.621,A -85,B 0,C 180,E1 -12426.478,E2 -12426.478} C_VEL
LIN {X 0,Y 376.109,Z 303.635,A -85,B 0,C 180,E1 -12429.682,E2 -12429.682} C_VEL
LIN {X 0,Y 376.08,Z 303.637,A -85,B 0,C 180,E1 -12433.658,E2 -12433.658} C_VEL
LIN {X 0,Y 376.036,Z 303.642,A -85,B 0,C 180,E1 -12437.608,E2 -12437.608} C_VEL
LIN {X 0,Y 375.97,Z 303.649,A -85,B 0,C 180,E1 -12440.833,E2 -12440.833} C_VEL
LIN {X 0,Y 375.979,Z 303.654,A -85,B 0,C 180,E1 -12444.283,E2 -12444.283} C_VEL
LIN {X 0,Y 376.011,Z 303.647,A -85,B 0,C 180,E1 -12446.653,E2 -12446.653} C_VEL
LIN {X 0,Y 375.963,Z 303.65,A -85,B 0,C 180,E1 -12449.08,E2 -12449.08} C_VEL
LIN {X 0,Y 375.942,Z 303.656,A -85,B 0,C 180,E1 -12452.829,E2 -12452.829} C_VEL
LIN {X 0,Y 375.95,Z 303.651,A -85,B 0,C 180,E1 -12455.417,E2 -12455.417} C_VEL
LIN {X 0,Y 375.929,Z 303.656,A -85,B 0,C 180,E1 -12458.264,E2 -12458.264} C_VEL
LIN {X 0,Y 375.913,Z 303.656,A -85,B 0,C 180,E1 -12461.599,E2 -12461.599} C_VEL
LIN {X 0,Y 375.921,Z 303.66,A -85,B 0,C 180,E1 -12464.732,E2 -12464.732} C_VEL
LIN {X 0,Y 375.92,Z 303.655,A -85,B 0,C 180,E1 -12467.7,E2 -12467.7} C_VEL
LIN {X 0,Y 375.931,Z 303.655,A -85,B 0,C 180,E1 -12470.535,E2 -12470.535} C_VEL
LIN {X 0,Y 375.959,Z 303.652,A -85,B 0,C 180,E1 -12473.497,E2 -12473.497} C_VEL
LIN {X 0,Y 375.957,Z 303.65,A -85,B 0,C 180,E1 -12475.89,E2 -12475.89} C_VEL
LIN {X 0,Y 375.959,Z 303.652,A -85,B 0,C 180,E1 -12479.688,E2 -12479.688} C_VEL
LIN {X 0,Y 375.915,Z 303.655,A -85,B 0,C 180,E1 -12482.136,E2 -12482.136} C_VEL
LIN {X 0,Y 375.958,Z 303.654,A -85,B 0,C 180,E1 -12485.717,E2 -12485.717} C_VEL
LIN {X 0,Y 375.998,Z 303.648,A -85,B 0,C 180,E1 -12489.199,E2 -12489.199} C_VEL
LIN {X 0,Y 376.033,Z 303.64,A -85,B 0,C 180,E1 -12492.601,E2 -12492.601} C_VEL
LIN {X 0,Y 376.09,Z 303.634,A -85,B 0,C 180,E1 -12496.344,E2 -12496.344} C_VEL
LIN {X 0,Y 376.106,Z 303.636,A -85,B 0,C 180,E1 -12500.319,E2 -12500.319} C_VEL
LIN {X 0,Y 376.117,Z 303.709,A -85,B 0,C 180,E1 -12500.93,E2 -12500.93} C_VEL
LIN {X 0,Y 377.887,Z 313.74,A -85,B 0,C 180,E1 -12503.46,E2 -12503.46} C_VEL
LIN {X 0,Y 378.039,Z 314.489,A -85,B 0,C 180,E1 -12503.546,E2 -12503.546} C_VEL
LIN {X 0,Y 382.577,Z 338.28,A -85,B 0,C 180,E1 -12504.222,E2 -12504.222} C_VEL
LIN {X 0,Y 381.267,Z 421.483,A -85,B 0,C 180,E1 -12505.802,E2 -12505.802} C_VEL
LIN {X 0,Y 380.796,Z 434.995,A -85,B 0,C 180,E1 -12506.277,E2 -12506.277} C_VEL
LIN {X 0,Y 380.254,Z 447.741,A -85,B 0,C 180,E1 -12506.949,E2 -12506.949} C_VEL
LIN {X 0,Y 379.591,Z 458.777,A -85,B 0,C 180,E1 -12507.733,E2 -12507.733} C_VEL
LIN {X 0,Y 378.775,Z 470.467,A -85,B 0,C 180,E1 -12508.805,E2 -12508.805} C_VEL
LIN {X 0,Y 377.894,Z 480.875,A -85,B 0,C 180,E1 -12510.001,E2 -12510.001} C_VEL
LIN {X 0,Y 377.028,Z 490.25,A -85,B 0,C 180,E1 -12511.336,E2 -12511.336} C_VEL
LIN {X 0,Y 376.236,Z 499.288,A -85,B 0,C 180,E1 -12512.945,E2 -12512.945} C_VEL
LIN {X 0,Y 375.644,Z 506.573,A -85,B 0,C 180,E1 -12514.561,E2 -12514.561} C_VEL
LIN {X 0,Y 375.309,Z 511.498,A -85,B 0,C 180,E1 -12515.912,E2 -12515.912} C_VEL
LIN {X 0,Y 374.964,Z 516.294,A -85,B 0,C 180,E1 -12517.54,E2 -12517.54} C_VEL
LIN {X 0,Y 374.698,Z 519.976,A -85,B 0,C 180,E1 -12519.174,E2 -12519.174} C_VEL
LIN {X 0,Y 374.515,Z 522.631,A -85,B 0,C 180,E1 -12520.817,E2 -12520.817} C_VEL
LIN {X 0,Y 374.445,Z 524.42,A -85,B 0,C 180,E1 -12522.604,E2 -12522.604} C_VEL
LIN {X 0,Y 374.387,Z 525.073,A -85,B 0,C 180,E1 -12524.125,E2 -12524.125} C_VEL
LIN {X 0,Y 374.394,Z 525.062,A -85,B 0,C 180,E1 -12525.237,E2 -12525.237} C_VEL
LIN {X 0,Y 374.497,Z 524.287,A -85,B 0,C 180,E1 -12526.844,E2 -12526.844} C_VEL
LIN {X 0,Y 374.528,Z 523.914,A -85,B 0,C 180,E1 -12527.281,E2 -12527.281} C_VEL
LIN {X 0,Y 373.974,Z 523.064,A -85,B 0,C 180,E1 -12528.173,E2 -12528.173} C_VEL
LIN {X 0,Y 371.377,Z 521.234,A -85,B 0,C 180,E1 -12529.618,E2 -12529.618} C_VEL
LIN {X 0,Y 369.235,Z 519.254,A -85,B 0,C 180,E1 -12530.766,E2 -12530.766} C_VEL
LIN {X 0,Y 368.432,Z 517.386,A -85,B 0,C 180,E1 -12531.632,E2 -12531.632} C_VEL
LIN {X 0,Y 368.43,Z 516.667,A -85,B 0,C 180,E1 -12531.919,E2 -12531.919} C_VEL
LIN {X 0,Y 369.162,Z 510.687,A -85,B 0,C 180,E1 -12533.962,E2 -12533.962} C_VEL
LIN {X 0,Y 369.97,Z 504.435,A -85,B 0,C 180,E1 -12535.605,E2 -12535.605} C_VEL
LIN {X 0,Y 371.049,Z 496.237,A -85,B 0,C 180,E1 -12537.313,E2 -12537.313} C_VEL
LIN {X 0,Y 372.124,Z 487.446,A -85,B 0,C 180,E1 -12538.79,E2 -12538.79} C_VEL
LIN {X 0,Y 373.232,Z 478.73,A -85,B 0,C 180,E1 -12539.981,E2 -12539.981} C_VEL
LIN {X 0,Y 374.343,Z 468.899,A -85,B 0,C 180,E1 -12541.084,E2 -12541.084} C_VEL
LIN {X 0,Y 375.43,Z 457.69,A -85,B 0,C 180,E1 -12542.085,E2 -12542.085} C_VEL
LIN {X 0,Y 376.354,Z 445.146,A -85,B 0,C 180,E1 -12542.948,E2 -12542.948} C_VEL
LIN {X 0,Y 377.058,Z 432.983,A -85,B 0,C 180,E1 -12543.557,E2 -12543.557} C_VEL
LIN {X 0,Y 377.539,Z 419.794,A -85,B 0,C 180,E1 -12543.985,E2 -12543.985} C_VEL
LIN {X 0,Y 379.194,Z 339.896,A -85,B 0,C 180,E1 -12545.535,E2 -12545.535} C_VEL
LIN {X 0,Y 375.825,Z 325.561,A -85,B 0,C 180,E1 -12546.079,E2 -12546.079} C_VEL
LIN {X 0,Y 371.22,Z 314.551,A -85,B 0,C 180,E1 -12546.676,E2 -12546.676} C_VEL
LIN {X 0,Y 368.931,Z 304.528,A -85,B 0,C 180,E1 -12549.478,E2 -12549.478} C_VEL
LIN {X 0,Y 368.888,Z 304.537,A -85,B 0,C 180,E1 -12553.304,E2 -12553.304} C_VEL
LIN {X 0,Y 368.887,Z 304.53,A -85,B 0,C 180,E1 -12556.696,E2 -12556.696} C_VEL
LIN {X 0,Y 368.914,Z 304.531,A -85,B 0,C 180,E1 -12559.643,E2 -12559.643} C_VEL
LIN {X 0,Y 368.904,Z 304.535,A -85,B 0,C 180,E1 -12563.144,E2 -12563.144} C_VEL
LIN {X 0,Y 368.898,Z 304.534,A -85,B 0,C 180,E1 -12566.462,E2 -12566.462} C_VEL
LIN {X 0,Y 368.931,Z 304.528,A -85,B 0,C 180,E1 -12569.046,E2 -12569.046} C_VEL
LIN {X 0,Y 368.981,Z 304.522,A -85,B 0,C 180,E1 -12571.564,E2 -12571.564} C_VEL
LIN {X 0,Y 369.001,Z 304.517,A -85,B 0,C 180,E1 -12574.02,E2 -12574.02} C_VEL
LIN {X 0,Y 368.933,Z 304.526,A -85,B 0,C 180,E1 -12577.605,E2 -12577.605} C_VEL
LIN {X 0,Y 368.983,Z 304.516,A -85,B 0,C 180,E1 -12581.107,E2 -12581.107} C_VEL
LIN {X 0,Y 368.999,Z 304.516,A -85,B 0,C 180,E1 -12584.535,E2 -12584.535} C_VEL
LIN {X 0,Y 369.006,Z 304.52,A -85,B 0,C 180,E1 -12587.907,E2 -12587.907} C_VEL
LIN {X 0,Y 369.23,Z 304.488,A -85,B 0,C 180,E1 -12591.801,E2 -12591.801} C_VEL
LIN {X 0,Y 369.143,Z 304.496,A -85,B 0,C 180,E1 -12594.537,E2 -12594.537} C_VEL
LIN {X 0,Y 369.317,Z 304.48,A -85,B 0,C 180,E1 -12597.819,E2 -12597.819} C_VEL
LIN {X 0,Y 369.457,Z 304.455,A -85,B 0,C 180,E1 -12600,E2 -12600} C_VEL
LIN {X 0,Y 369.317,Z 304.475,A -85,B 0,C 180,E1 -12602.181,E2 -12602.181} C_VEL
LIN {X 0,Y 369.207,Z 304.486,A -85,B 0,C 180,E1 -12606.558,E2 -12606.558} C_VEL
LIN {X 0,Y 369.138,Z 304.5,A -85,B 0,C 180,E1 -12608.761,E2 -12608.761} C_VEL
LIN {X 0,Y 369.004,Z 304.509,A -85,B 0,C 180,E1 -12612.093,E2 -12612.093} C_VEL
LIN {X 0,Y 368.998,Z 304.512,A -85,B 0,C 180,E1 -12615.465,E2 -12615.465} C_VEL
LIN {X 0,Y 368.983,Z 304.522,A -85,B 0,C 180,E1 -12618.893,E2 -12618.893} C_VEL
LIN {X 0,Y 368.926,Z 304.525,A -85,B 0,C 180,E1 -12622.396,E2 -12622.396} C_VEL
LIN {X 0,Y 369.001,Z 304.509,A -85,B 0,C 180,E1 -12625.98,E2 -12625.98} C_VEL
LIN {X 0,Y 368.962,Z 304.523,A -85,B 0,C 180,E1 -12628.811,E2 -12628.811} C_VEL
LIN {X 0,Y 368.899,Z 304.531,A -85,B 0,C 180,E1 -12632.238,E2 -12632.238} C_VEL
LIN {X 0,Y 368.93,Z 304.527,A -85,B 0,C 180,E1 -12635.001,E2 -12635.001} C_VEL
LIN {X 0,Y 368.909,Z 304.53,A -85,B 0,C 180,E1 -12638.64,E2 -12638.64} C_VEL
LIN {X 0,Y 368.883,Z 304.535,A -85,B 0,C 180,E1 -12642.009,E2 -12642.009} C_VEL
LIN {X 0,Y 368.882,Z 304.538,A -85,B 0,C 180,E1 -12645.176,E2 -12645.176} C_VEL
LIN {X 0,Y 368.884,Z 304.534,A -85,B 0,C 180,E1 -12648.177,E2 -12648.177} C_VEL
LIN {X 0,Y 368.908,Z 304.525,A -85,B 0,C 180,E1 -12651.36,E2 -12651.36} C_VEL
LIN {X 0,Y 368.939,Z 304.529,A -85,B 0,C 180,E1 -12655.146,E2 -12655.146} C_VEL
LIN {X 0,Y 368.923,Z 304.662,A -85,B 0,C 180,E1 -12659.01,E2 -12659.01} C_VEL
LIN {X 0,Y 371.691,Z 316.056,A -85,B 0,C 180,E1 -12662.03,E2 -12662.03} C_VEL
LIN {X 0,Y 373.511,Z 325.323,A -85,B 0,C 180,E1 -12664.356,E2 -12664.356} C_VEL
LIN {X 0,Y 373.143,Z 330.49,A -85,B 0,C 180,E1 -12665.52,E2 -12665.52} C_VEL
LIN {X 0,Y 372.264,Z 339.318,A -85,B 0,C 180,E1 -12667.473,E2 -12667.473} C_VEL
LIN {X 0,Y 376.237,Z 358.828,A -85,B 0,C 180,E1 -12668.18,E2 -12668.18} C_VEL
LIN {X 0,Y 378.517,Z 373.479,A -85,B 0,C 180,E1 -12668.646,E2 -12668.646} C_VEL
LIN {X 0,Y 377.26,Z 445.326,A -85,B 0,C 180,E1 -12670.053,E2 -12670.053} C_VEL
LIN {X 0,Y 376.629,Z 458.94,A -85,B 0,C 180,E1 -12670.479,E2 -12670.479} C_VEL
LIN {X 0,Y 375.707,Z 471.615,A -85,B 0,C 180,E1 -12671.104,E2 -12671.104} C_VEL
LIN {X 0,Y 374.585,Z 484.279,A -85,B 0,C 180,E1 -12671.966,E2 -12671.966} C_VEL
LIN {X 0,Y 373.243,Z 496.146,A -85,B 0,C 180,E1 -12673.03,E2 -12673.03} C_VEL
LIN {X 0,Y 372.016,Z 506.739,A -85,B 0,C 180,E1 -12674.242,E2 -12674.242} C_VEL
LIN {X 0,Y 370.995,Z 515.951,A -85,B 0,C 180,E1 -12675.547,E2 -12675.547} C_VEL
LIN {X 0,Y 369.902,Z 524.876,A -85,B 0,C 180,E1 -12677.1,E2 -12677.1} C_VEL
LIN {X 0,Y 368.884,Z 532.438,A -85,B 0,C 180,E1 -12678.738,E2 -12678.738} C_VEL
LIN {X 0,Y 368.158,Z 539.453,A -85,B 0,C 180,E1 -12680.661,E2 -12680.661} C_VEL
LIN {X 0,Y 367.73,Z 544.121,A -85,B 0,C 180,E1 -12682.311,E2 -12682.311} C_VEL
LIN {X 0,Y 367.507,Z 547.664,A -85,B 0,C 180,E1 -12683.946,E2 -12683.946} C_VEL
LIN {X 0,Y 367.457,Z 550.275,A -85,B 0,C 180,E1 -12685.612,E2 -12685.612} C_VEL
LIN {X 0,Y 367.381,Z 551.495,A -85,B 0,C 180,E1 -12686.709,E2 -12686.709} C_VEL
LIN {X 0,Y 367.396,Z 552.279,A -85,B 0,C 180,E1 -12687.807,E2 -12687.807} C_VEL
LIN {X 0,Y 367.457,Z 552.667,A -85,B 0,C 180,E1 -12688.903,E2 -12688.903} C_VEL
LIN {X 0,Y 367.504,Z 552.668,A -85,B 0,C 180,E1 -12689.999,E2 -12689.999} C_VEL
LIN {X 0,Y 367.487,Z 552.28,A -85,B 0,C 180,E1 -12691.095,E2 -12691.095} C_VEL
LIN {X 0,Y 367.425,Z 551.459,A -85,B 0,C 180,E1 -12692.192,E2 -12692.192} C_VEL
LIN {X 0,Y 367.488,Z 548.574,A -85,B 0,C 180,E1 -12694.386,E2 -12694.386} C_VEL
LIN {X 0,Y 367.514,Z 545.18,A -85,B 0,C 180,E1 -12696.065,E2 -12696.065} C_VEL
LIN {X 0,Y 367.693,Z 540.829,A -85,B 0,C 180,E1 -12697.688,E2 -12697.688} C_VEL
LIN {X 0,Y 368.017,Z 535.197,A -85,B 0,C 180,E1 -12699.341,E2 -12699.341} C_VEL
LIN {X 0,Y 368.501,Z 528.146,A -85,B 0,C 180,E1 -12700.994,E2 -12700.994} C_VEL
LIN {X 0,Y 369.357,Z 519.307,A -85,B 0,C 180,E1 -12702.639,E2 -12702.639} C_VEL
LIN {X 0,Y 370.252,Z 509.248,A -85,B 0,C 180,E1 -12704.145,E2 -12704.145} C_VEL
LIN {X 0,Y 371.059,Z 498.962,A -85,B 0,C 180,E1 -12705.376,E2 -12705.376} C_VEL
LIN {X 0,Y 371.917,Z 487.532,A -85,B 0,C 180,E1 -12706.465,E2 -12706.465} C_VEL
LIN {X 0,Y 372.829,Z 475.68,A -85,B 0,C 180,E1 -12707.341,E2 -12707.341} C_VEL
LIN {X 0,Y 373.606,Z 462.63,A -85,B 0,C 180,E1 -12708.046,E2 -12708.046} C_VEL
LIN {X 0,Y 374.184,Z 449.776,A -85,B 0,C 180,E1 -12708.513,E2 -12708.513} C_VEL
LIN {X 0,Y 374.874,Z 411.859,A -85,B 0,C 180,E1 -12709.27,E2 -12709.27} C_VEL
LIN {X 0,Y 375.242,Z 372.009,A -85,B 0,C 180,E1 -12710.04,E2 -12710.04} C_VEL
LIN {X 0,Y 370.779,Z 339.932,A -85,B 0,C 180,E1 -12710.897,E2 -12710.897} C_VEL
LIN {X 0,Y 372.112,Z 323.033,A -85,B 0,C 180,E1 -12714.55,E2 -12714.55} C_VEL
LIN {X 0,Y 371.794,Z 318.657,A -85,B 0,C 180,E1 -12715.539,E2 -12715.539} C_VEL
LIN {X 0,Y 369.006,Z 304.54,A -85,B 0,C 180,E1 -12718.896,E2 -12718.896} C_VEL
LIN {X 0,Y 368.896,Z 304.535,A -85,B 0,C 180,E1 -12722.237,E2 -12722.237} C_VEL
LIN {X 0,Y 368.926,Z 304.526,A -85,B 0,C 180,E1 -12725,E2 -12725} C_VEL
LIN {X 0,Y 368.902,Z 304.532,A -85,B 0,C 180,E1 -12728.639,E2 -12728.639} C_VEL
LIN {X 0,Y 368.876,Z 304.535,A -85,B 0,C 180,E1 -12732.008,E2 -12732.008} C_VEL
LIN {X 0,Y 368.876,Z 304.533,A -85,B 0,C 180,E1 -12735.175,E2 -12735.175} C_VEL
LIN {X 0,Y 368.878,Z 304.534,A -85,B 0,C 180,E1 -12738.177,E2 -12738.177} C_VEL
LIN {X 0,Y 368.904,Z 304.529,A -85,B 0,C 180,E1 -12741.358,E2 -12741.358} C_VEL
LIN {X 0,Y 368.93,Z 304.528,A -85,B 0,C 180,E1 -12745.146,E2 -12745.146} C_VEL
LIN {X 0,Y 368.922,Z 304.531,A -85,B 0,C 180,E1 -12749.046,E2 -12749.046} C_VEL
LIN {X 0,Y 368.979,Z 304.52,A -85,B 0,C 180,E1 -12751.564,E2 -12751.564} C_VEL
LIN {X 0,Y 368.949,Z 304.527,A -85,B 0,C 180,E1 -12755.224,E2 -12755.224} C_VEL
LIN {X 0,Y 368.929,Z 304.531,A -85,B 0,C 180,E1 -12758.973,E2 -12758.973} C_VEL
LIN {X 0,Y 368.982,Z 304.519,A -85,B 0,C 180,E1 -12762.257,E2 -12762.257} C_VEL
LIN {X 0,Y 369.028,Z 304.513,A -85,B 0,C 180,E1 -12766.227,E2 -12766.227} C_VEL
LIN {X 0,Y 369.059,Z 304.51,A -85,B 0,C 180,E1 -12770.132,E2 -12770.132} C_VEL
LIN {X 0,Y 369.179,Z 304.494,A -85,B 0,C 180,E1 -12772.342,E2 -12772.342} C_VEL
LIN {X 0,Y 369.135,Z 304.5,A -85,B 0,C 180,E1 -12774.537,E2 -12774.537} C_VEL
LIN {X 0,Y 369.309,Z 304.483,A -85,B 0,C 180,E1 -12777.819,E2 -12777.819} C_VEL
LIN {X 0,Y 369.449,Z 304.464,A -85,B 0,C 180,E1 -12780,E2 -12780} C_VEL
LIN {X 0,Y 369.31,Z 304.48,A -85,B 0,C 180,E1 -12782.181,E2 -12782.181} C_VEL
LIN {X 0,Y 369.163,Z 304.497,A -85,B 0,C 180,E1 -12786.559,E2 -12786.559} C_VEL
LIN {X 0,Y 369.058,Z 304.516,A -85,B 0,C 180,E1 -12789.869,E2 -12789.869} C_VEL
LIN {X 0,Y 369.028,Z 304.517,A -85,B 0,C 180,E1 -12793.773,E2 -12793.773} C_VEL
LIN {X 0,Y 368.993,Z 304.52,A -85,B 0,C 180,E1 -12797.769,E2 -12797.769} C_VEL
LIN {X 0,Y 368.901,Z 304.529,A -85,B 0,C 180,E1 -12801.222,E2 -12801.222} C_VEL
LIN {X 0,Y 368.945,Z 304.526,A -85,B 0,C 180,E1 -12804.776,E2 -12804.776} C_VEL
LIN {X 0,Y 368.96,Z 304.522,A -85,B 0,C 180,E1 -12807.204,E2 -12807.204} C_VEL
LIN {X 0,Y 368.911,Z 304.528,A -85,B 0,C 180,E1 -12809.691,E2 -12809.691} C_VEL
LIN {X 0,Y 368.89,Z 304.532,A -85,B 0,C 180,E1 -12813.044,E2 -12813.044} C_VEL
LIN {X 0,Y 368.91,Z 304.53,A -85,B 0,C 180,E1 -12816.198,E2 -12816.198} C_VEL
LIN {X 0,Y 368.868,Z 304.537,A -85,B 0,C 180,E1 -12818.958,E2 -12818.958} C_VEL
LIN {X 0,Y 368.865,Z 304.534,A -85,B 0,C 180,E1 -12822.009,E2 -12822.009} C_VEL
LIN {X 0,Y 368.873,Z 304.536,A -85,B 0,C 180,E1 -12825.177,E2 -12825.177} C_VEL
LIN {X 0,Y 368.864,Z 304.534,A -85,B 0,C 180,E1 -12828.177,E2 -12828.177} C_VEL
LIN {X 0,Y 368.873,Z 304.536,A -85,B 0,C 180,E1 -12831.367,E2 -12831.367} C_VEL
LIN {X 0,Y 368.933,Z 304.532,A -85,B 0,C 180,E1 -12835.148,E2 -12835.148} C_VEL
LIN {X 0,Y 368.91,Z 304.532,A -85,B 0,C 180,E1 -12839.046,E2 -12839.046} C_VEL
LIN {X 0,Y 368.904,Z 304.533,A -85,B 0,C 180,E1 -12841.559,E2 -12841.559} C_VEL
LIN {X 0,Y 368.912,Z 304.532,A -85,B 0,C 180,E1 -12845.223,E2 -12845.223} C_VEL
LIN {X 0,Y 368.909,Z 304.528,A -85,B 0,C 180,E1 -12848.78,E2 -12848.78} C_VEL
LIN {X 0,Y 368.991,Z 304.518,A -85,B 0,C 180,E1 -12852.258,E2 -12852.258} C_VEL
LIN {X 0,Y 369.038,Z 304.513,A -85,B 0,C 180,E1 -12856.229,E2 -12856.229} C_VEL
LIN {X 0,Y 369.086,Z 304.511,A -85,B 0,C 180,E1 -12860.617,E2 -12860.617} C_VEL
LIN {X 0,Y 369.291,Z 305.603,A -85,B 0,C 180,E1 -12860.968,E2 -12860.968} C_VEL
LIN {X 0,Y 370.853,Z 314.389,A -85,B 0,C 180,E1 -12863.199,E2 -12863.199} C_VEL
LIN {X 0,Y 374.585,Z 332.424,A -85,B 0,C 180,E1 -12863.737,E2 -12863.737} C_VEL
LIN {X 0,Y 375.721,Z 338.746,A -85,B 0,C 180,E1 -12863.916,E2 -12863.916} C_VEL
LIN {X 0,Y 374.419,Z 422.393,A -85,B 0,C 180,E1 -12865.544,E2 -12865.544} C_VEL
LIN {X 0,Y 373.938,Z 435.787,A -85,B 0,C 180,E1 -12866.032,E2 -12866.032} C_VEL
LIN {X 0,Y 373.414,Z 447.228,A -85,B 0,C 180,E1 -12866.645,E2 -12866.645} C_VEL
LIN {X 0,Y 372.734,Z 458.368,A -85,B 0,C 180,E1 -12867.434,E2 -12867.434} C_VEL
LIN {X 0,Y 371.903,Z 470.072,A -85,B 0,C 180,E1 -12868.512,E2 -12868.512} C_VEL
LIN {X 0,Y 371.007,Z 480.588,A -85,B 0,C 180,E1 -12869.729,E2 -12869.729} C_VEL
